LIN {X 0.214,Y -702.984,Z 640.438,A 0.000,B 0.000,C 90.000,E1 294.847} C_DIS
LIN {X -0.283,Y -702.330,Z 640.438,A 0.000,B 0.000,C 90.000,E1 294.771} C_DIS
LIN {X 0.270,Y -699.025,Z 640.435,A 0.000,B 0.000,C 90.000,E1 294.259} C_DIS
LIN {X 0.118,Y -697.927,Z 640.434,A 0.000,B 0.000,C 90.000,E1 294.155} C_DIS
LIN {X 0.250,Y -696.247,Z 640.434,A 0.000,B 0.000,C 90.000,E1 294.027} C_DIS
LIN {X 0.435,Y -691.769,Z 640.433,A 0.000,B 0.000,C 90.000,E1 293.823} C_DIS
LIN {X 0.326,Y -685.920,Z 640.432,A 0.000,B 0.000,C 90.000,E1 293.643} C_DIS
LIN {X -0.028,Y -681.507,Z 640.431,A 0.000,B 0.000,C 90.000,E1 293.567} C_DIS
LIN {X -0.084,Y -673.236,Z 640.430,A 0.000,B 0.000,C 90.000,E1 293.462} C_DIS
LIN {X 0.101,Y -666.043,Z 640.430,A 0.000,B 0.000,C 90.000,E1 293.387} C_DIS
LIN {X 0.093,Y -649.725,Z 640.429,A 0.000,B 0.000,C 90.000,E1 293.153} C_DIS
LIN {X -0.148,Y -639.864,Z 640.428,A 0.000,B 0.000,C 90.000,E1 293.003} C_DIS
LIN {X 0.048,Y -630.020,Z 640.427,A 0.000,B 0.000,C 90.000,E1 292.770} C_DIS
LIN {X -0.345,Y -616.725,Z 640.425,A 0.000,B 0.000,C 90.000,E1 292.461} C_DIS
LIN {X 0.086,Y -589.337,Z 640.420,A 0.000,B 0.000,C 90.000,E1 291.589} C_DIS
LIN {X -0.163,Y -576.913,Z 640.418,A 0.000,B 0.000,C 90.000,E1 291.227} C_DIS
LIN {X -0.001,Y -564.499,Z 640.416,A 0.000,B 0.000,C 90.000,E1 290.844} C_DIS
LIN {X 0.289,Y -559.704,Z 640.415,A 0.000,B 0.000,C 90.000,E1 290.610} C_DIS
LIN {X 0.143,Y -556.813,Z 640.414,A 0.000,B 0.000,C 90.000,E1 290.429} C_DIS
LIN {X 0.112,Y -556.775,Z 640.414,A 0.000,B 0.000,C 90.000,E1 290.429} C_DIS
LIN {X -0.163,Y -556.015,Z 640.412,A 0.000,B 0.000,C 90.000,E1 290.248} C_DIS
LIN {X 0.014,Y -555.587,Z 640.410,A 0.000,B 0.000,C 90.000,E1 289.812} C_DIS
LIN {X -0.233,Y -555.561,Z 640.404,A 0.000,B 0.000,C 90.000,E1 288.725} C_DIS
LIN {X -0.215,Y -555.366,Z 640.396,A 0.000,B 0.000,C 90.000,E1 287.330} C_DIS
LIN {X -0.115,Y -555.080,Z 640.390,A 0.000,B 0.000,C 90.000,E1 286.205} C_DIS
LIN {X 0.258,Y -554.527,Z 640.382,A 0.000,B 0.000,C 90.000,E1 284.773} C_DIS
LIN {X -0.065,Y -553.860,Z 640.375,A 0.000,B 0.000,C 90.000,E1 283.411} C_DIS
LIN {X 0.136,Y -552.938,Z 640.365,A 0.000,B 0.000,C 90.000,E1 281.715} C_DIS
LIN {X 0.079,Y -552.458,Z 640.359,A 0.000,B 0.000,C 90.000,E1 280.602} C_DIS
LIN {X 0.264,Y -551.690,Z 640.348,A 0.000,B 0.000,C 90.000,E1 278.624} C_DIS
LIN {X -0.277,Y -550.949,Z 640.337,A 0.000,B 0.000,C 90.000,E1 276.720} C_DIS
LIN {X 0.258,Y -550.396,Z 640.326,A 0.000,B 0.000,C 90.000,E1 274.702} C_DIS
LIN {X 0.000,Y -550.065,Z 640.319,A 0.000,B 0.000,C 90.000,E1 273.326} C_DIS
LIN {X -0.182,Y -549.599,Z 640.309,A 0.000,B 0.000,C 90.000,E1 271.661} C_DIS
LIN {X 0.139,Y -549.034,Z 640.300,A 0.000,B 0.000,C 90.000,E1 269.943} C_DIS
LIN {X -0.153,Y -548.291,Z 640.292,A 0.000,B 0.000,C 90.000,E1 268.568} C_DIS
LIN {X 0.101,Y -547.676,Z 640.284,A 0.000,B 0.000,C 90.000,E1 267.135} C_DIS
LIN {X -0.168,Y -546.950,Z 640.276,A 0.000,B 0.000,C 90.000,E1 265.755} C_DIS
LIN {X 0.100,Y -545.943,Z 640.269,A 0.000,B 0.000,C 90.000,E1 264.318} C_DIS
LIN {X -0.140,Y -544.897,Z 640.261,A 0.000,B 0.000,C 90.000,E1 262.932} C_DIS
LIN {X 0.057,Y -543.716,Z 640.254,A 0.000,B 0.000,C 90.000,E1 261.781} C_DIS
LIN {X 0.013,Y -541.556,Z 640.243,A 0.000,B 0.000,C 90.000,E1 259.803} C_DIS
LIN {X -0.159,Y -540.004,Z 640.234,A 0.000,B 0.000,C 90.000,E1 258.117} C_DIS
LIN {X -0.015,Y -538.115,Z 640.221,A 0.000,B 0.000,C 90.000,E1 255.825} C_DIS
LIN {X -0.019,Y -537.132,Z 640.215,A 0.000,B 0.000,C 90.000,E1 254.685} C_DIS
LIN {X -0.173,Y -535.984,Z 640.209,A 0.000,B 0.000,C 90.000,E1 253.559} C_DIS
LIN {X -0.230,Y -533.804,Z 640.196,A 0.000,B 0.000,C 90.000,E1 251.275} C_DIS
LIN {X 0.193,Y -532.904,Z 640.191,A 0.000,B 0.000,C 90.000,E1 250.369} C_DIS
LIN {X -0.201,Y -531.346,Z 640.185,A 0.000,B 0.000,C 90.000,E1 249.263} C_DIS
LIN {X 0.066,Y -529.285,Z 640.177,A 0.000,B 0.000,C 90.000,E1 247.794} C_DIS
LIN {X -0.176,Y -527.436,Z 640.170,A 0.000,B 0.000,C 90.000,E1 246.666} C_DIS
LIN {X -0.130,Y -525.978,Z 640.165,A 0.000,B 0.000,C 90.000,E1 245.793} C_DIS
LIN {X 0.280,Y -523.709,Z 640.159,A 0.000,B 0.000,C 90.000,E1 244.588} C_DIS
LIN {X -0.047,Y -521.275,Z 640.153,A 0.000,B 0.000,C 90.000,E1 243.461} C_DIS
LIN {X 0.187,Y -518.199,Z 640.144,A 0.000,B 0.000,C 90.000,E1 241.975} C_DIS
LIN {X -0.092,Y -515.078,Z 640.136,A 0.000,B 0.000,C 90.000,E1 240.539} C_DIS
LIN {X 0.182,Y -512.332,Z 640.130,A 0.000,B 0.000,C 90.000,E1 239.331} C_DIS
LIN {X -0.046,Y -508.136,Z 640.120,A 0.000,B 0.000,C 90.000,E1 237.582} C_DIS
LIN {X 0.015,Y -504.589,Z 640.112,A 0.000,B 0.000,C 90.000,E1 236.087} C_DIS
LIN {X -0.013,Y -501.554,Z 640.105,A 0.000,B 0.000,C 90.000,E1 234.895} C_DIS
LIN {X -0.083,Y -498.368,Z 640.098,A 0.000,B 0.000,C 90.000,E1 233.703} C_DIS
LIN {X 0.072,Y -491.532,Z 640.083,A 0.000,B 0.000,C 90.000,E1 230.964} C_DIS
LIN {X 0.058,Y -487.091,Z 640.073,A 0.000,B 0.000,C 90.000,E1 229.138} C_DIS
LIN {X -0.113,Y -481.191,Z 640.059,A 0.000,B 0.000,C 90.000,E1 226.701} C_DIS
LIN {X 0.054,Y -478.156,Z 640.053,A 0.000,B 0.000,C 90.000,E1 225.445} C_DIS
LIN {X 0.278,Y -474.467,Z 640.044,A 0.000,B 0.000,C 90.000,E1 223.866} C_DIS
LIN {X -0.233,Y -470.885,Z 640.035,A 0.000,B 0.000,C 90.000,E1 222.366} C_DIS
LIN {X 0.140,Y -465.420,Z 640.021,A 0.000,B 0.000,C 90.000,E1 219.806} C_DIS
LIN {X -0.098,Y -461.340,Z 640.011,A 0.000,B 0.000,C 90.000,E1 217.935} C_DIS
LIN {X -0.151,Y -456.212,Z 639.997,A 0.000,B 0.000,C 90.000,E1 215.391} C_DIS
LIN {X -0.138,Y -453.326,Z 639.988,A 0.000,B 0.000,C 90.000,E1 213.785} C_DIS
LIN {X -0.101,Y -448.042,Z 639.971,A 0.000,B 0.000,C 90.000,E1 210.875} C_DIS
LIN {X 0.105,Y -444.631,Z 639.961,A 0.000,B 0.000,C 90.000,E1 208.899} C_DIS
LIN {X 0.018,Y -441.087,Z 639.950,A 0.000,B 0.000,C 90.000,E1 206.950} C_DIS
LIN {X -0.030,Y -438.709,Z 639.943,A 0.000,B 0.000,C 90.000,E1 205.643} C_DIS
LIN {X 0.136,Y -435.079,Z 639.932,A 0.000,B 0.000,C 90.000,E1 203.643} C_DIS
LIN {X 0.014,Y -432.764,Z 639.924,A 0.000,B 0.000,C 90.000,E1 202.333} C_DIS
LIN {X 0.086,Y -428.719,Z 639.911,A 0.000,B 0.000,C 90.000,E1 199.993} C_DIS
LIN {X 0.156,Y -424.805,Z 639.898,A 0.000,B 0.000,C 90.000,E1 197.638} C_DIS
LIN {X -0.188,Y -421.615,Z 639.887,A 0.000,B 0.000,C 90.000,E1 195.662} C_DIS
LIN {X 0.035,Y -418.916,Z 639.878,A 0.000,B 0.000,C 90.000,E1 193.939} C_DIS
LIN {X 0.058,Y -415.763,Z 639.866,A 0.000,B 0.000,C 90.000,E1 191.895} C_DIS
LIN {X 0.058,Y -412.228,Z 639.853,A 0.000,B 0.000,C 90.000,E1 189.500} C_DIS
LIN {X 0.200,Y -410.259,Z 639.845,A 0.000,B 0.000,C 90.000,E1 188.106} C_DIS
LIN {X -0.151,Y -406.790,Z 639.832,A 0.000,B 0.000,C 90.000,E1 185.739} C_DIS
LIN {X 0.128,Y -403.391,Z 639.816,A 0.000,B 0.000,C 90.000,E1 182.922} C_DIS
LIN {X -0.036,Y -398.663,Z 639.789,A 0.000,B 0.000,C 90.000,E1 178.051} C_DIS
LIN {X 0.172,Y -396.253,Z 639.766,A 0.000,B 0.000,C 90.000,E1 173.799} C_DIS
LIN {X -0.114,Y -395.651,Z 639.754,A 0.000,B 0.000,C 90.000,E1 171.724} C_DIS
LIN {X 0.123,Y -395.202,Z 639.740,A 0.000,B 0.000,C 90.000,E1 169.218} C_DIS
LIN {X 0.025,Y -395.157,Z 639.721,A 0.000,B 0.000,C 90.000,E1 165.700} C_DIS
LIN {X -0.195,Y -395.441,Z 639.705,A 0.000,B 0.000,C 90.000,E1 162.906} C_DIS
LIN {X 0.192,Y -395.870,Z 639.693,A 0.000,B 0.000,C 90.000,E1 160.732} C_DIS
LIN {X -0.020,Y -396.318,Z 639.681,A 0.000,B 0.000,C 90.000,E1 158.646} C_DIS
LIN {X -0.012,Y -396.971,Z 639.668,A 0.000,B 0.000,C 90.000,E1 156.177} C_DIS
LIN {X -0.041,Y -397.593,Z 639.654,A 0.000,B 0.000,C 90.000,E1 153.717} C_DIS
LIN {X 0.066,Y -398.150,Z 639.642,A 0.000,B 0.000,C 90.000,E1 151.591} C_DIS
LIN {X -0.197,Y -398.673,Z 639.633,A 0.000,B 0.000,C 90.000,E1 149.871} C_DIS
LIN {X -0.023,Y -399.254,Z 639.621,A 0.000,B 0.000,C 90.000,E1 147.740} C_DIS
LIN {X 0.140,Y -400.146,Z 639.607,A 0.000,B 0.000,C 90.000,E1 145.261} C_DIS
LIN {X -0.212,Y -401.026,Z 639.596,A 0.000,B 0.000,C 90.000,E1 143.210} C_DIS
LIN {X -0.176,Y -401.737,Z 639.586,A 0.000,B 0.000,C 90.000,E1 141.457} C_DIS
LIN {X 0.132,Y -402.461,Z 639.576,A 0.000,B 0.000,C 90.000,E1 139.666} C_DIS
LIN {X 0.149,Y -403.113,Z 639.566,A 0.000,B 0.000,C 90.000,E1 137.919} C_DIS
LIN {X -0.008,Y -403.916,Z 639.555,A 0.000,B 0.000,C 90.000,E1 135.850} C_DIS
LIN {X -0.042,Y -404.957,Z 639.541,A 0.000,B 0.000,C 90.000,E1 133.419} C_DIS
LIN {X 0.105,Y -406.638,Z 639.526,A 0.000,B 0.000,C 90.000,E1 130.620} C_DIS
LIN {X 0.078,Y -407.304,Z 639.522,A 0.000,B 0.000,C 90.000,E1 129.930} C_DIS
LIN {X 0.029,Y -408.620,Z 639.517,A 0.000,B 0.000,C 90.000,E1 129.072} C_DIS
LIN {X 0.015,Y -410.546,Z 639.513,A 0.000,B 0.000,C 90.000,E1 128.382} C_DIS
LIN {X -0.069,Y -411.560,Z 639.512,A 0.000,B 0.000,C 90.000,E1 128.222} C_DIS
LIN {X -0.162,Y -413.181,Z 639.510,A 0.000,B 0.000,C 90.000,E1 127.890} C_DIS
LIN {X 0.099,Y -416.926,Z 639.508,A 0.000,B 0.000,C 90.000,E1 127.443} C_DIS
LIN {X -0.118,Y -420.836,Z 639.506,A 0.000,B 0.000,C 90.000,E1 127.156} C_DIS
LIN {X 0.057,Y -442.467,Z 639.499,A 0.000,B 0.000,C 90.000,E1 125.724} C_DIS
LIN {X -0.069,Y -450.784,Z 639.496,A 0.000,B 0.000,C 90.000,E1 125.231} C_DIS
LIN {X -0.113,Y -460.538,Z 639.492,A 0.000,B 0.000,C 90.000,E1 124.612} C_DIS
LIN {X 0.212,Y -473.139,Z 639.487,A 0.000,B 0.000,C 90.000,E1 123.706} C_DIS
LIN {X -0.040,Y -480.978,Z 639.484,A 0.000,B 0.000,C 90.000,E1 123.166} C_DIS
LIN {X -0.212,Y -488.438,Z 639.481,A 0.000,B 0.000,C 90.000,E1 122.625} C_DIS
LIN {X -0.011,Y -496.000,Z 639.478,A 0.000,B 0.000,C 90.000,E1 122.005} C_DIS
LIN {X -0.106,Y -505.725,Z 639.473,A 0.000,B 0.000,C 90.000,E1 121.209} C_DIS
LIN {X -0.173,Y -512.904,Z 639.470,A 0.000,B 0.000,C 90.000,E1 120.590} C_DIS
LIN {X -0.071,Y -518.358,Z 639.467,A 0.000,B 0.000,C 90.000,E1 120.079} C_DIS
LIN {X -0.102,Y -524.925,Z 639.464,A 0.000,B 0.000,C 90.000,E1 119.461} C_DIS
LIN {X 0.099,Y -531.758,Z 639.460,A 0.000,B 0.000,C 90.000,E1 118.771} C_DIS
LIN {X 0.053,Y -536.831,Z 639.457,A 0.000,B 0.000,C 90.000,E1 118.231} C_DIS
LIN {X -0.113,Y -541.360,Z 639.454,A 0.000,B 0.000,C 90.000,E1 117.719} C_DIS
LIN {X -0.071,Y -546.495,Z 639.450,A 0.000,B 0.000,C 90.000,E1 117.052} C_DIS
LIN {X -0.077,Y -550.302,Z 639.447,A 0.000,B 0.000,C 90.000,E1 116.488} C_DIS
LIN {X -0.163,Y -554.583,Z 639.443,A 0.000,B 0.000,C 90.000,E1 115.796} C_DIS
LIN {X -0.078,Y -559.013,Z 639.439,A 0.000,B 0.000,C 90.000,E1 114.951} C_DIS
LIN {X -0.189,Y -562.959,Z 639.434,A 0.000,B 0.000,C 90.000,E1 114.131} C_DIS
LIN {X 0.258,Y -566.594,Z 639.429,A 0.000,B 0.000,C 90.000,E1 113.259} C_DIS
LIN {X -0.001,Y -569.978,Z 639.425,A 0.000,B 0.000,C 90.000,E1 112.461} C_DIS
LIN {X 0.140,Y -573.938,Z 639.419,A 0.000,B 0.000,C 90.000,E1 111.354} C_DIS
LIN {X 0.333,Y -575.783,Z 639.416,A 0.000,B 0.000,C 90.000,E1 110.791} C_DIS
LIN {X 0.172,Y -578.288,Z 639.411,A 0.000,B 0.000,C 90.000,E1 109.993} C_DIS
LIN {X 0.227,Y -581.303,Z 639.405,A 0.000,B 0.000,C 90.000,E1 108.906} C_DIS
LIN {X -0.067,Y -583.345,Z 639.401,A 0.000,B 0.000,C 90.000,E1 108.127} C_DIS
LIN {X -0.266,Y -586.358,Z 639.393,A 0.000,B 0.000,C 90.000,E1 106.804} C_DIS
LIN {X -0.076,Y -591.364,Z 639.381,A 0.000,B 0.000,C 90.000,E1 104.647} C_DIS
LIN {X 0.099,Y -595.831,Z 639.371,A 0.000,B 0.000,C 90.000,E1 102.771} C_DIS
LIN {X -0.203,Y -598.908,Z 639.364,A 0.000,B 0.000,C 90.000,E1 101.478} C_DIS
LIN {X 0.017,Y -602.053,Z 639.356,A 0.000,B 0.000,C 90.000,E1 100.141} C_DIS
LIN {X -0.301,Y -605.007,Z 639.349,A 0.000,B 0.000,C 90.000,E1 98.859} C_DIS
LIN {X 0.295,Y -607.255,Z 639.343,A 0.000,B 0.000,C 90.000,E1 97.757} C_DIS
LIN {X -0.039,Y -609.837,Z 639.336,A 0.000,B 0.000,C 90.000,E1 96.486} C_DIS
LIN {X -0.124,Y -612.554,Z 639.327,A 0.000,B 0.000,C 90.000,E1 94.935} C_DIS
LIN {X 0.176,Y -614.578,Z 639.320,A 0.000,B 0.000,C 90.000,E1 93.612} C_DIS
LIN {X -0.146,Y -616.328,Z 639.313,A 0.000,B 0.000,C 90.000,E1 92.350} C_DIS
LIN {X -0.133,Y -617.527,Z 639.307,A 0.000,B 0.000,C 90.000,E1 91.318} C_DIS
LIN {X -0.112,Y -618.745,Z 639.299,A 0.000,B 0.000,C 90.000,E1 89.771} C_DIS
LIN {X -0.085,Y -619.350,Z 639.293,A 0.000,B 0.000,C 90.000,E1 88.740} C_DIS
LIN {X -0.033,Y -619.644,Z 639.287,A 0.000,B 0.000,C 90.000,E1 87.707} C_DIS
LIN {X -0.321,Y -619.669,Z 639.283,A 0.000,B 0.000,C 90.000,E1 86.963} C_DIS
LIN {X -0.224,Y -619.534,Z 639.277,A 0.000,B 0.000,C 90.000,E1 85.927} C_DIS
LIN {X -0.168,Y -619.186,Z 639.272,A 0.000,B 0.000,C 90.000,E1 84.894} C_DIS
LIN {X 0.233,Y -618.474,Z 639.264,A 0.000,B 0.000,C 90.000,E1 83.571} C_DIS
LIN {X -0.292,Y -617.789,Z 639.259,A 0.000,B 0.000,C 90.000,E1 82.591} C_DIS
LIN {X 0.114,Y -617.072,Z 639.254,A 0.000,B 0.000,C 90.000,E1 81.781} C_DIS
LIN {X 0.268,Y -615.828,Z 639.249,A 0.000,B 0.000,C 90.000,E1 80.735} C_DIS
LIN {X 0.163,Y -614.044,Z 639.242,A 0.000,B 0.000,C 90.000,E1 79.454} C_DIS
LIN {X 0.025,Y -611.983,Z 639.234,A 0.000,B 0.000,C 90.000,E1 78.173} C_DIS
LIN {X -0.025,Y -609.699,Z 639.227,A 0.000,B 0.000,C 90.000,E1 76.881} C_DIS
LIN {X 0.140,Y -607.779,Z 639.221,A 0.000,B 0.000,C 90.000,E1 75.825} C_DIS
LIN {X 0.161,Y -605.161,Z 639.214,A 0.000,B 0.000,C 90.000,E1 74.519} C_DIS
LIN {X -0.169,Y -602.830,Z 639.208,A 0.000,B 0.000,C 90.000,E1 73.504} C_DIS
LIN {X -0.058,Y -599.843,Z 639.201,A 0.000,B 0.000,C 90.000,E1 72.181} C_DIS
LIN {X 0.295,Y -597.192,Z 639.195,A 0.000,B 0.000,C 90.000,E1 71.094} C_DIS
LIN {X 0.046,Y -594.117,Z 639.189,A 0.000,B 0.000,C 90.000,E1 70.061} C_DIS
LIN {X 0.074,Y -591.600,Z 639.185,A 0.000,B 0.000,C 90.000,E1 69.263} C_DIS
LIN {X 0.078,Y -588.849,Z 639.180,A 0.000,B 0.000,C 90.000,E1 68.465} C_DIS
LIN {X -0.072,Y -584.716,Z 639.174,A 0.000,B 0.000,C 90.000,E1 67.411} C_DIS
LIN {X -0.277,Y -580.359,Z 639.169,A 0.000,B 0.000,C 90.000,E1 66.357} C_DIS
LIN {X 0.063,Y -574.233,Z 639.161,A 0.000,B 0.000,C 90.000,E1 64.973} C_DIS
LIN {X 0.268,Y -571.589,Z 639.158,A 0.000,B 0.000,C 90.000,E1 64.409} C_DIS
LIN {X -0.063,Y -568.759,Z 639.155,A 0.000,B 0.000,C 90.000,E1 63.896} C_DIS
LIN {X 0.005,Y -564.884,Z 639.151,A 0.000,B 0.000,C 90.000,E1 63.204} C_DIS
LIN {X -0.112,Y -561.591,Z 639.148,A 0.000,B 0.000,C 90.000,E1 62.666} C_DIS
LIN {X 0.097,Y -557.022,Z 639.144,A 0.000,B 0.000,C 90.000,E1 61.975} C_DIS
LIN {X -0.062,Y -553.002,Z 639.141,A 0.000,B 0.000,C 90.000,E1 61.435} C_DIS
LIN {X 0.088,Y -549.418,Z 639.139,A 0.000,B 0.000,C 90.000,E1 61.001} C_DIS
LIN {X 0.124,Y -547.052,Z 639.137,A 0.000,B 0.000,C 90.000,E1 60.717} C_DIS
LIN {X -0.069,Y -543.497,Z 639.135,A 0.000,B 0.000,C 90.000,E1 60.333} C_DIS
LIN {X 0.302,Y -538.237,Z 639.132,A 0.000,B 0.000,C 90.000,E1 59.793} C_DIS
LIN {X -0.209,Y -533.738,Z 639.130,A 0.000,B 0.000,C 90.000,E1 59.459} C_DIS
LIN {X -0.199,Y -527.676,Z 639.128,A 0.000,B 0.000,C 90.000,E1 58.997} C_DIS
LIN {X 0.158,Y -521.319,Z 639.125,A 0.000,B 0.000,C 90.000,E1 58.535} C_DIS
LIN {X 0.023,Y -516.351,Z 639.124,A 0.000,B 0.000,C 90.000,E1 58.250} C_DIS
LIN {X 0.258,Y -506.211,Z 639.121,A 0.000,B 0.000,C 90.000,E1 57.661} C_DIS
LIN {X -0.156,Y -482.576,Z 639.114,A 0.000,B 0.000,C 90.000,E1 56.501} C_DIS
LIN {X 0.027,Y -460.468,Z 639.108,A 0.000,B 0.000,C 90.000,E1 55.341} C_DIS
LIN {X 0.094,Y -438.216,Z 639.101,A 0.000,B 0.000,C 90.000,E1 54.116} C_DIS
LIN {X 0.050,Y -438.150,Z 639.101,A 0.000,B 0.000,C 90.000,E1 54.116} C_DIS
LIN {X -0.079,Y -431.839,Z 639.083,A 0.000,B 0.000,C 90.000,E1 51.009} C_DIS
LIN {X 0.180,Y -431.143,Z 639.082,A 0.000,B 0.000,C 90.000,E1 50.642} C_DIS
LIN {X 0.111,Y -423.698,Z 639.064,A 0.000,B 0.000,C 90.000,E1 47.472} C_DIS
LIN {X 0.080,Y -424.089,Z 639.057,A 0.000,B 0.000,C 90.000,E1 46.296} C_DIS
LIN {X -0.206,Y -424.329,Z 639.052,A 0.000,B 0.000,C 90.000,E1 45.324} C_DIS
LIN {X -0.052,Y -424.762,Z 639.037,A 0.000,B 0.000,C 90.000,E1 42.609} C_DIS
LIN {X -0.275,Y -425.406,Z 639.026,A 0.000,B 0.000,C 90.000,E1 40.620} C_DIS
LIN {X 0.064,Y -426.388,Z 639.012,A 0.000,B 0.000,C 90.000,E1 38.222} C_DIS
LIN {X -0.003,Y -427.318,Z 639.001,A 0.000,B 0.000,C 90.000,E1 36.217} C_DIS
LIN {X -0.167,Y -428.037,Z 638.994,A 0.000,B 0.000,C 90.000,E1 34.898} C_DIS
LIN {X -0.094,Y -428.902,Z 638.983,A 0.000,B 0.000,C 90.000,E1 32.880} C_DIS
LIN {X -0.104,Y -429.733,Z 638.971,A 0.000,B 0.000,C 90.000,E1 30.875} C_DIS
LIN {X -0.096,Y -430.417,Z 638.962,A 0.000,B 0.000,C 90.000,E1 29.205} C_DIS
LIN {X 0.085,Y -431.164,Z 638.953,A 0.000,B 0.000,C 90.000,E1 27.513} C_DIS
LIN {X -0.104,Y -432.164,Z 638.942,A 0.000,B 0.000,C 90.000,E1 25.540} C_DIS
LIN {X 0.122,Y -433.288,Z 638.931,A 0.000,B 0.000,C 90.000,E1 23.515} C_DIS
LIN {X 0.029,Y -434.557,Z 638.920,A 0.000,B 0.000,C 90.000,E1 21.535} C_DIS
LIN {X -0.020,Y -435.592,Z 638.911,A 0.000,B 0.000,C 90.000,E1 19.885} C_DIS
LIN {X 0.188,Y -436.754,Z 638.899,A 0.000,B 0.000,C 90.000,E1 17.873} C_DIS
LIN {X -0.149,Y -438.145,Z 638.887,A 0.000,B 0.000,C 90.000,E1 15.607} C_DIS
LIN {X 0.109,Y -440.016,Z 638.872,A 0.000,B 0.000,C 90.000,E1 12.939} C_DIS
LIN {X -0.030,Y -441.896,Z 638.859,A 0.000,B 0.000,C 90.000,E1 10.658} C_DIS
LIN {X 0.067,Y -444.666,Z 638.843,A 0.000,B 0.000,C 90.000,E1 7.701} C_DIS
LIN {X 0.111,Y -446.688,Z 638.832,A 0.000,B 0.000,C 90.000,E1 5.739} C_DIS
LIN {X 0.180,Y -450.113,Z 638.816,A 0.000,B 0.000,C 90.000,E1 2.808} C_DIS
LIN {X -0.199,Y -452.588,Z 638.805,A 0.000,B 0.000,C 90.000,E1 0.917} C_DIS
LIN {X 0.163,Y -456.504,Z 638.790,A 0.000,B 0.000,C 90.000,E1 358.165} C_DIS
LIN {X 0.204,Y -459.105,Z 638.781,A 0.000,B 0.000,C 90.000,E1 356.560} C_DIS
LIN {X 0.055,Y -462.306,Z 638.770,A 0.000,B 0.000,C 90.000,E1 354.666} C_DIS
LIN {X 0.063,Y -465.626,Z 638.760,A 0.000,B 0.000,C 90.000,E1 352.761} C_DIS
LIN {X 0.217,Y -468.922,Z 638.749,A 0.000,B 0.000,C 90.000,E1 350.849} C_DIS
LIN {X -0.132,Y -471.112,Z 638.742,A 0.000,B 0.000,C 90.000,E1 349.634} C_DIS
LIN {X 0.148,Y -474.860,Z 638.730,A 0.000,B 0.000,C 90.000,E1 347.409} C_DIS
LIN {X 0.020,Y -479.405,Z 638.716,A 0.000,B 0.000,C 90.000,E1 344.936} C_DIS
LIN {X -0.192,Y -484.083,Z 638.703,A 0.000,B 0.000,C 90.000,E1 342.489} C_DIS
LIN {X 0.159,Y -487.675,Z 638.692,A 0.000,B 0.000,C 90.000,E1 340.604} C_DIS
LIN {X 0.111,Y -490.671,Z 638.684,A 0.000,B 0.000,C 90.000,E1 339.082} C_DIS
LIN {X 0.252,Y -493.055,Z 638.677,A 0.000,B 0.000,C 90.000,E1 337.847} C_DIS
LIN {X -0.074,Y -494.653,Z 638.672,A 0.000,B 0.000,C 90.000,E1 336.975} C_DIS
LIN {X -0.281,Y -497.144,Z 638.664,A 0.000,B 0.000,C 90.000,E1 335.485} C_DIS
LIN {X 0.031,Y -499.972,Z 638.654,A 0.000,B 0.000,C 90.000,E1 333.640} C_DIS
LIN {X -0.044,Y -502.754,Z 638.644,A 0.000,B 0.000,C 90.000,E1 331.847} C_DIS
LIN {X 0.198,Y -508.652,Z 638.625,A 0.000,B 0.000,C 90.000,E1 328.535} C_DIS
LIN {X 0.054,Y -510.798,Z 638.620,A 0.000,B 0.000,C 90.000,E1 327.661} C_DIS
LIN {X 0.298,Y -512.682,Z 638.617,A 0.000,B 0.000,C 90.000,E1 327.041} C_DIS
LIN {X -0.155,Y -515.106,Z 638.614,A 0.000,B 0.000,C 90.000,E1 326.501} C_DIS
LIN {X 0.306,Y -517.597,Z 638.611,A 0.000,B 0.000,C 90.000,E1 326.008} C_DIS
LIN {X 0.062,Y -520.974,Z 638.609,A 0.000,B 0.000,C 90.000,E1 325.595} C_DIS
LIN {X 0.192,Y -523.917,Z 638.607,A 0.000,B 0.000,C 90.000,E1 325.261} C_DIS
LIN {X 0.257,Y -530.298,Z 638.604,A 0.000,B 0.000,C 90.000,E1 324.689} C_DIS
LIN {X -0.225,Y -547.687,Z 638.596,A 0.000,B 0.000,C 90.000,E1 323.336} C_DIS
LIN {X -0.048,Y -556.154,Z 638.592,A 0.000,B 0.000,C 90.000,E1 322.603} C_DIS
LIN {X 0.167,Y -567.400,Z 638.587,A 0.000,B 0.000,C 90.000,E1 321.618} C_DIS
LIN {X 0.174,Y -579.786,Z 638.581,A 0.000,B 0.000,C 90.000,E1 320.517} C_DIS
LIN {X 0.169,Y -590.603,Z 638.575,A 0.000,B 0.000,C 90.000,E1 319.542} C_DIS
LIN {X 0.208,Y -599.582,Z 638.571,A 0.000,B 0.000,C 90.000,E1 318.690} C_DIS
LIN {X 0.147,Y -603.451,Z 638.569,A 0.000,B 0.000,C 90.000,E1 318.324} C_DIS
LIN {X -0.384,Y -611.958,Z 638.564,A 0.000,B 0.000,C 90.000,E1 317.472} C_DIS
LIN {X 0.089,Y -617.498,Z 638.560,A 0.000,B 0.000,C 90.000,E1 316.782} C_DIS
LIN {X 0.044,Y -620.550,Z 638.558,A 0.000,B 0.000,C 90.000,E1 316.419} C_DIS
LIN {X 0.378,Y -626.351,Z 638.554,A 0.000,B 0.000,C 90.000,E1 315.648} C_DIS
LIN {X 0.004,Y -632.030,Z 638.550,A 0.000,B 0.000,C 90.000,E1 314.919} C_DIS
LIN {X -0.319,Y -637.451,Z 638.545,A 0.000,B 0.000,C 90.000,E1 314.190} C_DIS
LIN {X -0.209,Y -644.470,Z 638.540,A 0.000,B 0.000,C 90.000,E1 313.176} C_DIS
LIN {X 0.071,Y -648.686,Z 638.536,A 0.000,B 0.000,C 90.000,E1 312.528} C_DIS
LIN {X -0.016,Y -651.957,Z 638.534,A 0.000,B 0.000,C 90.000,E1 312.043} C_DIS
LIN {X -0.098,Y -656.684,Z 638.529,A 0.000,B 0.000,C 90.000,E1 311.310} C_DIS
LIN {X -0.158,Y -660.324,Z 638.526,A 0.000,B 0.000,C 90.000,E1 310.701} C_DIS
LIN {X 0.267,Y -664.285,Z 638.522,A 0.000,B 0.000,C 90.000,E1 309.930} C_DIS
LIN {X -0.197,Y -666.771,Z 638.519,A 0.000,B 0.000,C 90.000,E1 309.483} C_DIS
LIN {X -0.142,Y -670.151,Z 638.515,A 0.000,B 0.000,C 90.000,E1 308.749} C_DIS
LIN {X 0.062,Y -674.214,Z 638.510,A 0.000,B 0.000,C 90.000,E1 307.764} C_DIS
LIN {X 0.195,Y -676.940,Z 638.506,A 0.000,B 0.000,C 90.000,E1 307.030} C_DIS
LIN {X -0.046,Y -680.209,Z 638.501,A 0.000,B 0.000,C 90.000,E1 306.091} C_DIS
LIN {X 0.303,Y -683.353,Z 638.495,A 0.000,B 0.000,C 90.000,E1 305.105} C_DIS
LIN {X -0.056,Y -687.653,Z 638.487,A 0.000,B 0.000,C 90.000,E1 303.706} C_DIS
LIN {X 0.001,Y -690.328,Z 638.482,A 0.000,B 0.000,C 90.000,E1 302.752} C_DIS
LIN {X -0.265,Y -693.426,Z 638.475,A 0.000,B 0.000,C 90.000,E1 301.592} C_DIS
LIN {X 0.100,Y -695.821,Z 638.470,A 0.000,B 0.000,C 90.000,E1 300.620} C_DIS
LIN {X -0.094,Y -698.544,Z 638.464,A 0.000,B 0.000,C 90.000,E1 299.461} C_DIS
LIN {X 0.351,Y -700.491,Z 638.458,A 0.000,B 0.000,C 90.000,E1 298.487} C_DIS
LIN {X -0.123,Y -702.298,Z 638.453,A 0.000,B 0.000,C 90.000,E1 297.590} C_DIS
LIN {X 0.092,Y -703.480,Z 638.449,A 0.000,B 0.000,C 90.000,E1 296.873} C_DIS
LIN {X 0.001,Y -704.295,Z 638.445,A 0.000,B 0.000,C 90.000,E1 296.181} C_DIS
LIN {X -0.059,Y -704.501,Z 638.443,A 0.000,B 0.000,C 90.000,E1 295.720} C_DIS
LIN {X 0.228,Y -704.340,Z 638.442,A 0.000,B 0.000,C 90.000,E1 295.463} C_DIS
LIN {X -0.138,Y -703.279,Z 638.439,A 0.000,B 0.000,C 90.000,E1 295.027} C_DIS
LIN {X 0.146,Y -702.359,Z 638.438,A 0.000,B 0.000,C 90.000,E1 294.771} C_DIS
LIN {X -0.227,Y -699.016,Z 638.435,A 0.000,B 0.000,C 90.000,E1 294.335} C_DIS
LIN {X -0.093,Y -698.007,Z 638.435,A 0.000,B 0.000,C 90.000,E1 294.207} C_DIS
LIN {X 0.040,Y -696.495,Z 638.434,A 0.000,B 0.000,C 90.000,E1 294.079} C_DIS
LIN {X 0.332,Y -694.302,Z 638.433,A 0.000,B 0.000,C 90.000,E1 293.951} C_DIS
LIN {X -0.173,Y -689.748,Z 638.432,A 0.000,B 0.000,C 90.000,E1 293.823} C_DIS
LIN {X -0.084,Y -685.927,Z 638.432,A 0.000,B 0.000,C 90.000,E1 293.695} C_DIS
LIN {X -0.003,Y -681.958,Z 638.431,A 0.000,B 0.000,C 90.000,E1 293.590} C_DIS
LIN {X 0.058,Y -672.967,Z 638.430,A 0.000,B 0.000,C 90.000,E1 293.462} C_DIS
LIN {X 0.228,Y -665.855,Z 638.430,A 0.000,B 0.000,C 90.000,E1 293.387} C_DIS
LIN {X -0.375,Y -649.556,Z 638.429,A 0.000,B 0.000,C 90.000,E1 293.206} C_DIS
LIN {X -0.269,Y -639.725,Z 638.428,A 0.000,B 0.000,C 90.000,E1 293.025} C_DIS
LIN {X 0.175,Y -629.930,Z 638.427,A 0.000,B 0.000,C 90.000,E1 292.770} C_DIS
LIN {X -0.233,Y -616.602,Z 638.425,A 0.000,B 0.000,C 90.000,E1 292.461} C_DIS
LIN {X -0.195,Y -596.132,Z 638.421,A 0.000,B 0.000,C 90.000,E1 291.844} C_DIS
LIN {X -0.051,Y -578.637,Z 638.418,A 0.000,B 0.000,C 90.000,E1 291.280} C_DIS
LIN {X -0.103,Y -564.298,Z 638.416,A 0.000,B 0.000,C 90.000,E1 290.865} C_DIS
LIN {X -0.169,Y -559.577,Z 638.415,A 0.000,B 0.000,C 90.000,E1 290.663} C_DIS
LIN {X 0.132,Y -556.796,Z 638.414,A 0.000,B 0.000,C 90.000,E1 290.429} C_DIS
LIN {X 0.097,Y -556.769,Z 638.414,A 0.000,B 0.000,C 90.000,E1 290.429} C_DIS
LIN {X -0.262,Y -555.974,Z 638.412,A 0.000,B 0.000,C 90.000,E1 290.248} C_DIS
LIN {X 0.212,Y -555.621,Z 638.410,A 0.000,B 0.000,C 90.000,E1 289.812} C_DIS
LIN {X -0.052,Y -555.663,Z 638.404,A 0.000,B 0.000,C 90.000,E1 288.725} C_DIS
LIN {X -0.032,Y -555.489,Z 638.396,A 0.000,B 0.000,C 90.000,E1 287.330} C_DIS
LIN {X 0.070,Y -555.179,Z 638.390,A 0.000,B 0.000,C 90.000,E1 286.205} C_DIS
LIN {X 0.178,Y -554.783,Z 638.384,A 0.000,B 0.000,C 90.000,E1 285.079} C_DIS
LIN {X 0.000,Y -554.133,Z 638.376,A 0.000,B 0.000,C 90.000,E1 283.703} C_DIS
LIN {X 0.079,Y -553.373,Z 638.368,A 0.000,B 0.000,C 90.000,E1 282.299} C_DIS
LIN {X 0.272,Y -552.563,Z 638.359,A 0.000,B 0.000,C 90.000,E1 280.602} C_DIS
LIN {X -0.086,Y -551.792,Z 638.348,A 0.000,B 0.000,C 90.000,E1 278.681} C_DIS
LIN {X -0.120,Y -551.132,Z 638.339,A 0.000,B 0.000,C 90.000,E1 277.004} C_DIS
LIN {X -0.186,Y -550.526,Z 638.328,A 0.000,B 0.000,C 90.000,E1 275.049} C_DIS
LIN {X 0.200,Y -550.101,Z 638.319,A 0.000,B 0.000,C 90.000,E1 273.326} C_DIS
LIN {X -0.052,Y -549.745,Z 638.311,A 0.000,B 0.000,C 90.000,E1 271.949} C_DIS
LIN {X -0.262,Y -549.195,Z 638.302,A 0.000,B 0.000,C 90.000,E1 270.286} C_DIS
LIN {X -0.051,Y -548.685,Z 638.295,A 0.000,B 0.000,C 90.000,E1 269.141} C_DIS
LIN {X -0.241,Y -547.751,Z 638.284,A 0.000,B 0.000,C 90.000,E1 267.192} C_DIS
LIN {X -0.040,Y -547.209,Z 638.278,A 0.000,B 0.000,C 90.000,E1 266.045} C_DIS
LIN {X 0.192,Y -546.471,Z 638.272,A 0.000,B 0.000,C 90.000,E1 264.894} C_DIS
LIN {X -0.016,Y -545.254,Z 638.262,A 0.000,B 0.000,C 90.000,E1 263.223} C_DIS
LIN {X 0.172,Y -544.484,Z 638.258,A 0.000,B 0.000,C 90.000,E1 262.356} C_DIS
LIN {X -0.019,Y -542.628,Z 638.248,A 0.000,B 0.000,C 90.000,E1 260.679} C_DIS
LIN {X 0.057,Y -540.175,Z 638.234,A 0.000,B 0.000,C 90.000,E1 258.117} C_DIS
LIN {X 0.205,Y -538.283,Z 638.221,A 0.000,B 0.000,C 90.000,E1 255.825} C_DIS
LIN {X 0.260,Y -537.008,Z 638.214,A 0.000,B 0.000,C 90.000,E1 254.393} C_DIS
LIN {X -0.169,Y -535.266,Z 638.204,A 0.000,B 0.000,C 90.000,E1 252.725} C_DIS
LIN {X 0.197,Y -533.637,Z 638.194,A 0.000,B 0.000,C 90.000,E1 250.967} C_DIS
LIN {X 0.117,Y -532.640,Z 638.190,A 0.000,B 0.000,C 90.000,E1 250.115} C_DIS
LIN {X 0.222,Y -531.059,Z 638.183,A 0.000,B 0.000,C 90.000,E1 248.954} C_DIS
LIN {X -0.194,Y -529.404,Z 638.177,A 0.000,B 0.000,C 90.000,E1 247.847} C_DIS
LIN {X 0.233,Y -527.074,Z 638.169,A 0.000,B 0.000,C 90.000,E1 246.357} C_DIS
LIN {X -0.207,Y -525.526,Z 638.164,A 0.000,B 0.000,C 90.000,E1 245.537} C_DIS
LIN {X 0.198,Y -523.203,Z 638.158,A 0.000,B 0.000,C 90.000,E1 244.332} C_DIS
LIN {X 0.240,Y -520.131,Z 638.149,A 0.000,B 0.000,C 90.000,E1 242.871} C_DIS
LIN {X 0.000,Y -517.027,Z 638.141,A 0.000,B 0.000,C 90.000,E1 241.435} C_DIS
LIN {X 0.051,Y -514.456,Z 638.135,A 0.000,B 0.000,C 90.000,E1 240.255} C_DIS
LIN {X -0.289,Y -512.397,Z 638.130,A 0.000,B 0.000,C 90.000,E1 239.410} C_DIS
LIN {X 0.185,Y -508.199,Z 638.120,A 0.000,B 0.000,C 90.000,E1 237.582} C_DIS
LIN {X 0.245,Y -504.596,Z 638.112,A 0.000,B 0.000,C 90.000,E1 236.087} C_DIS
LIN {X 0.217,Y -501.543,Z 638.105,A 0.000,B 0.000,C 90.000,E1 234.895} C_DIS
LIN {X 0.020,Y -497.617,Z 638.097,A 0.000,B 0.000,C 90.000,E1 233.417} C_DIS
LIN {X -0.235,Y -490.764,Z 638.082,A 0.000,B 0.000,C 90.000,E1 230.723} C_DIS
LIN {X 0.110,Y -486.303,Z 638.072,A 0.000,B 0.000,C 90.000,E1 228.852} C_DIS
LIN {X 0.107,Y -481.145,Z 638.060,A 0.000,B 0.000,C 90.000,E1 226.701} C_DIS
LIN {X -0.069,Y -478.105,Z 638.053,A 0.000,B 0.000,C 90.000,E1 225.486} C_DIS
LIN {X -0.075,Y -473.665,Z 638.042,A 0.000,B 0.000,C 90.000,E1 223.623} C_DIS
LIN {X -0.021,Y -470.824,Z 638.035,A 0.000,B 0.000,C 90.000,E1 222.366} C_DIS
LIN {X -0.069,Y -466.020,Z 638.023,A 0.000,B 0.000,C 90.000,E1 220.172} C_DIS
LIN {X -0.085,Y -463.308,Z 638.016,A 0.000,B 0.000,C 90.000,E1 218.910} C_DIS
LIN {X -0.165,Y -458.031,Z 638.002,A 0.000,B 0.000,C 90.000,E1 216.377} C_DIS
LIN {X 0.061,Y -453.259,Z 637.988,A 0.000,B 0.000,C 90.000,E1 213.785} C_DIS
LIN {X 0.093,Y -447.985,Z 637.972,A 0.000,B 0.000,C 90.000,E1 210.875} C_DIS
LIN {X -0.092,Y -444.575,Z 637.961,A 0.000,B 0.000,C 90.000,E1 208.949} C_DIS
LIN {X -0.186,Y -441.034,Z 637.950,A 0.000,B 0.000,C 90.000,E1 207.001} C_DIS
LIN {X -0.034,Y -438.667,Z 637.943,A 0.000,B 0.000,C 90.000,E1 205.668} C_DIS
LIN {X -0.085,Y -435.648,Z 637.933,A 0.000,B 0.000,C 90.000,E1 204.027} C_DIS
LIN {X 0.198,Y -432.731,Z 637.924,A 0.000,B 0.000,C 90.000,E1 202.333} C_DIS
LIN {X 0.267,Y -428.685,Z 637.911,A 0.000,B 0.000,C 90.000,E1 199.993} C_DIS
LIN {X -0.070,Y -424.793,Z 637.898,A 0.000,B 0.000,C 90.000,E1 197.692} C_DIS
LIN {X -0.010,Y -421.611,Z 637.887,A 0.000,B 0.000,C 90.000,E1 195.662} C_DIS
LIN {X -0.138,Y -418.429,Z 637.876,A 0.000,B 0.000,C 90.000,E1 193.647} C_DIS
LIN {X 0.010,Y -414.763,Z 637.862,A 0.000,B 0.000,C 90.000,E1 191.243} C_DIS
LIN {X -0.098,Y -411.330,Z 637.849,A 0.000,B 0.000,C 90.000,E1 188.859} C_DIS
LIN {X 0.037,Y -407.826,Z 637.836,A 0.000,B 0.000,C 90.000,E1 186.429} C_DIS
LIN {X -0.089,Y -403.840,Z 637.818,A 0.000,B 0.000,C 90.000,E1 183.326} C_DIS
LIN {X 0.135,Y -401.485,Z 637.807,A 0.000,B 0.000,C 90.000,E1 181.203} C_DIS
LIN {X 0.090,Y -398.442,Z 637.787,A 0.000,B 0.000,C 90.000,E1 177.707} C_DIS
LIN {X -0.118,Y -396.234,Z 637.764,A 0.000,B 0.000,C 90.000,E1 173.514} C_DIS
LIN {X 0.036,Y -395.656,Z 637.752,A 0.000,B 0.000,C 90.000,E1 171.376} C_DIS
LIN {X -0.113,Y -395.286,Z 637.738,A 0.000,B 0.000,C 90.000,E1 168.926} C_DIS
LIN {X -0.168,Y -395.283,Z 637.721,A 0.000,B 0.000,C 90.000,E1 165.755} C_DIS
LIN {X 0.000,Y -395.614,Z 637.705,A 0.000,B 0.000,C 90.000,E1 162.906} C_DIS
LIN {X 0.016,Y -396.015,Z 637.693,A 0.000,B 0.000,C 90.000,E1 160.786} C_DIS
LIN {X -0.026,Y -396.399,Z 637.684,A 0.000,B 0.000,C 90.000,E1 159.028} C_DIS
LIN {X 0.221,Y -396.837,Z 637.674,A 0.000,B 0.000,C 90.000,E1 157.230} C_DIS
LIN {X 0.113,Y -397.298,Z 637.664,A 0.000,B 0.000,C 90.000,E1 155.485} C_DIS
LIN {X 0.042,Y -397.903,Z 637.652,A 0.000,B 0.000,C 90.000,E1 153.384} C_DIS
LIN {X 0.163,Y -398.476,Z 637.641,A 0.000,B 0.000,C 90.000,E1 151.257} C_DIS
LIN {X -0.092,Y -398.987,Z 637.631,A 0.000,B 0.000,C 90.000,E1 149.537} C_DIS
LIN {X -0.247,Y -399.581,Z 637.619,A 0.000,B 0.000,C 90.000,E1 147.454} C_DIS
LIN {X 0.047,Y -400.347,Z 637.607,A 0.000,B 0.000,C 90.000,E1 145.308} C_DIS
LIN {X 0.031,Y -401.222,Z 637.596,A 0.000,B 0.000,C 90.000,E1 143.210} C_DIS
LIN {X 0.070,Y -401.927,Z 637.586,A 0.000,B 0.000,C 90.000,E1 141.457} C_DIS
LIN {X 0.121,Y -402.621,Z 637.576,A 0.000,B 0.000,C 90.000,E1 139.703} C_DIS
LIN {X 0.009,Y -403.118,Z 637.569,A 0.000,B 0.000,C 90.000,E1 138.324} C_DIS
LIN {X 0.131,Y -403.899,Z 637.557,A 0.000,B 0.000,C 90.000,E1 136.215} C_DIS
LIN {X -0.143,Y -404.580,Z 637.547,A 0.000,B 0.000,C 90.000,E1 134.514} C_DIS
LIN {X -0.011,Y -405.882,Z 637.532,A 0.000,B 0.000,C 90.000,E1 131.714} C_DIS
LIN {X 0.080,Y -407.193,Z 637.522,A 0.000,B 0.000,C 90.000,E1 129.967} C_DIS
LIN {X -0.110,Y -408.590,Z 637.516,A 0.000,B 0.000,C 90.000,E1 128.955} C_DIS
LIN {X -0.171,Y -410.677,Z 637.512,A 0.000,B 0.000,C 90.000,E1 128.177} C_DIS
LIN {X -0.012,Y -412.178,Z 637.510,A 0.000,B 0.000,C 90.000,E1 127.810} C_DIS
LIN {X -0.053,Y -412.711,Z 637.510,A 0.000,B 0.000,C 90.000,E1 127.729} C_DIS
LIN {X -0.055,Y -416.091,Z 637.507,A 0.000,B 0.000,C 90.000,E1 127.317} C_DIS
LIN {X 0.076,Y -419.643,Z 637.506,A 0.000,B 0.000,C 90.000,E1 126.996} C_DIS
LIN {X 0.061,Y -425.517,Z 637.503,A 0.000,B 0.000,C 90.000,E1 126.583} C_DIS
LIN {X -0.031,Y -447.482,Z 637.496,A 0.000,B 0.000,C 90.000,E1 125.231} C_DIS
LIN {X -0.117,Y -458.843,Z 637.492,A 0.000,B 0.000,C 90.000,E1 124.532} C_DIS
LIN {X -0.057,Y -471.653,Z 637.487,A 0.000,B 0.000,C 90.000,E1 123.658} C_DIS
LIN {X -0.048,Y -477.865,Z 637.485,A 0.000,B 0.000,C 90.000,E1 123.214} C_DIS
LIN {X -0.081,Y -487.034,Z 637.481,A 0.000,B 0.000,C 90.000,E1 122.546} C_DIS
LIN {X 0.113,Y -494.372,Z 637.478,A 0.000,B 0.000,C 90.000,E1 121.957} C_DIS
LIN {X -0.220,Y -498.431,Z 637.476,A 0.000,B 0.000,C 90.000,E1 121.671} C_DIS
LIN {X -0.090,Y -507.257,Z 637.472,A 0.000,B 0.000,C 90.000,E1 120.924} C_DIS
LIN {X 0.022,Y -512.960,Z 637.469,A 0.000,B 0.000,C 90.000,E1 120.413} C_DIS
LIN {X -0.004,Y -521.287,Z 637.465,A 0.000,B 0.000,C 90.000,E1 119.667} C_DIS
LIN {X 0.153,Y -530.711,Z 637.460,A 0.000,B 0.000,C 90.000,E1 118.743} C_DIS
LIN {X 0.120,Y -536.840,Z 637.456,A 0.000,B 0.000,C 90.000,E1 118.103} C_DIS
LIN {X -0.120,Y -541.711,Z 637.453,A 0.000,B 0.000,C 90.000,E1 117.564} C_DIS
LIN {X -0.159,Y -546.210,Z 637.450,A 0.000,B 0.000,C 90.000,E1 117.001} C_DIS
LIN {X 0.081,Y -550.146,Z 637.447,A 0.000,B 0.000,C 90.000,E1 116.411} C_DIS
LIN {X -0.008,Y -554.505,Z 637.443,A 0.000,B 0.000,C 90.000,E1 115.720} C_DIS
LIN {X 0.016,Y -558.920,Z 637.438,A 0.000,B 0.000,C 90.000,E1 114.899} C_DIS
LIN {X -0.095,Y -562.961,Z 637.434,A 0.000,B 0.000,C 90.000,E1 114.079} C_DIS
LIN {X 0.028,Y -565.491,Z 637.431,A 0.000,B 0.000,C 90.000,E1 113.515} C_DIS
LIN {X 0.103,Y -570.076,Z 637.425,A 0.000,B 0.000,C 90.000,E1 112.408} C_DIS
LIN {X -0.076,Y -574.110,Z 637.419,A 0.000,B 0.000,C 90.000,E1 111.334} C_DIS
LIN {X -0.091,Y -575.962,Z 637.416,A 0.000,B 0.000,C 90.000,E1 110.791} C_DIS
LIN {X 0.291,Y -578.551,Z 637.411,A 0.000,B 0.000,C 90.000,E1 109.939} C_DIS
LIN {X 0.155,Y -580.898,Z 637.406,A 0.000,B 0.000,C 90.000,E1 109.141} C_DIS
LIN {X -0.149,Y -583.019,Z 637.402,A 0.000,B 0.000,C 90.000,E1 108.362} C_DIS
LIN {X 0.132,Y -584.911,Z 637.398,A 0.000,B 0.000,C 90.000,E1 107.528} C_DIS
LIN {X -0.197,Y -588.585,Z 637.389,A 0.000,B 0.000,C 90.000,E1 105.953} C_DIS
LIN {X -0.223,Y -592.417,Z 637.380,A 0.000,B 0.000,C 90.000,E1 104.356} C_DIS
LIN {X -0.016,Y -596.955,Z 637.369,A 0.000,B 0.000,C 90.000,E1 102.479} C_DIS
LIN {X 0.306,Y -601.407,Z 637.359,A 0.000,B 0.000,C 90.000,E1 100.602} C_DIS
LIN {X -0.024,Y -604.446,Z 637.352,A 0.000,B 0.000,C 90.000,E1 99.321} C_DIS
LIN {X -0.038,Y -606.814,Z 637.346,A 0.000,B 0.000,C 90.000,E1 98.276} C_DIS
LIN {X 0.223,Y -609.485,Z 637.339,A 0.000,B 0.000,C 90.000,E1 96.947} C_DIS
LIN {X 0.195,Y -611.458,Z 637.333,A 0.000,B 0.000,C 90.000,E1 95.910} C_DIS
LIN {X -0.139,Y -613.677,Z 637.326,A 0.000,B 0.000,C 90.000,E1 94.645} C_DIS
LIN {X 0.134,Y -615.667,Z 637.319,A 0.000,B 0.000,C 90.000,E1 93.326} C_DIS
LIN {X 0.144,Y -617.051,Z 637.313,A 0.000,B 0.000,C 90.000,E1 92.293} C_DIS
LIN {X 0.166,Y -618.276,Z 637.307,A 0.000,B 0.000,C 90.000,E1 91.260} C_DIS
LIN {X -0.114,Y -619.308,Z 637.300,A 0.000,B 0.000,C 90.000,E1 90.000} C_DIS
LIN {X -0.078,Y -620.003,Z 637.294,A 0.000,B 0.000,C 90.000,E1 88.969} C_DIS
LIN {X 0.261,Y -620.274,Z 637.290,A 0.000,B 0.000,C 90.000,E1 88.167} C_DIS
LIN {X -0.297,Y -620.414,Z 637.284,A 0.000,B 0.000,C 90.000,E1 87.192} C_DIS
LIN {X 0.128,Y -620.213,Z 637.277,A 0.000,B 0.000,C 90.000,E1 85.869} C_DIS
LIN {X 0.192,Y -619.824,Z 637.271,A 0.000,B 0.000,C 90.000,E1 84.837} C_DIS
LIN {X -0.012,Y -619.107,Z 637.264,A 0.000,B 0.000,C 90.000,E1 83.571} C_DIS
LIN {X 0.084,Y -618.410,Z 637.259,A 0.000,B 0.000,C 90.000,E1 82.534} C_DIS
LIN {X -0.116,Y -617.658,Z 637.254,A 0.000,B 0.000,C 90.000,E1 81.781} C_DIS
LIN {X 0.046,Y -616.373,Z 637.249,A 0.000,B 0.000,C 90.000,E1 80.735} C_DIS
LIN {X -0.049,Y -614.549,Z 637.241,A 0.000,B 0.000,C 90.000,E1 79.454} C_DIS
LIN {X -0.178,Y -612.455,Z 637.234,A 0.000,B 0.000,C 90.000,E1 78.173} C_DIS
LIN {X 0.029,Y -610.616,Z 637.229,A 0.000,B 0.000,C 90.000,E1 77.117} C_DIS
LIN {X -0.047,Y -608.163,Z 637.221,A 0.000,B 0.000,C 90.000,E1 75.825} C_DIS
LIN {X -0.020,Y -605.479,Z 637.214,A 0.000,B 0.000,C 90.000,E1 74.519} C_DIS
LIN {X 0.234,Y -603.105,Z 637.208,A 0.000,B 0.000,C 90.000,E1 73.449} C_DIS
LIN {X -0.229,Y -600.059,Z 637.201,A 0.000,B 0.000,C 90.000,E1 72.181} C_DIS
LIN {X 0.129,Y -597.328,Z 637.195,A 0.000,B 0.000,C 90.000,E1 71.094} C_DIS
LIN {X -0.118,Y -594.152,Z 637.189,A 0.000,B 0.000,C 90.000,E1 70.061} C_DIS
LIN {X 0.141,Y -590.621,Z 637.183,A 0.000,B 0.000,C 90.000,E1 68.975} C_DIS
LIN {X 0.346,Y -587.719,Z 637.179,A 0.000,B 0.000,C 90.000,E1 68.156} C_DIS
LIN {X 0.179,Y -583.420,Z 637.173,A 0.000,B 0.000,C 90.000,E1 67.102} C_DIS
LIN {X 0.090,Y -580.041,Z 637.168,A 0.000,B 0.000,C 90.000,E1 66.305} C_DIS
LIN {X -0.111,Y -573.802,Z 637.161,A 0.000,B 0.000,C 90.000,E1 64.973} C_DIS
LIN {X -0.158,Y -568.895,Z 637.156,A 0.000,B 0.000,C 90.000,E1 64.024} C_DIS
LIN {X -0.087,Y -564.956,Z 637.152,A 0.000,B 0.000,C 90.000,E1 63.332} C_DIS
LIN {X 0.297,Y -561.626,Z 637.149,A 0.000,B 0.000,C 90.000,E1 62.743} C_DIS
LIN {X -0.044,Y -555.792,Z 637.144,A 0.000,B 0.000,C 90.000,E1 61.948} C_DIS
LIN {X 0.122,Y -552.731,Z 637.142,A 0.000,B 0.000,C 90.000,E1 61.513} C_DIS
LIN {X 0.072,Y -544.097,Z 637.136,A 0.000,B 0.000,C 90.000,E1 60.539} C_DIS
LIN {X -0.049,Y -542.807,Z 637.136,A 0.000,B 0.000,C 90.000,E1 60.411} C_DIS
LIN {X 0.115,Y -538.533,Z 637.133,A 0.000,B 0.000,C 90.000,E1 59.999} C_DIS
LIN {X 0.058,Y -534.575,Z 637.132,A 0.000,B 0.000,C 90.000,E1 59.665} C_DIS
LIN {X -0.202,Y -529.870,Z 637.130,A 0.000,B 0.000,C 90.000,E1 59.331} C_DIS
LIN {X 0.086,Y -526.782,Z 637.128,A 0.000,B 0.000,C 90.000,E1 59.076} C_DIS
LIN {X 0.171,Y -521.873,Z 637.127,A 0.000,B 0.000,C 90.000,E1 58.742} C_DIS
LIN {X 0.327,Y -515.153,Z 637.124,A 0.000,B 0.000,C 90.000,E1 58.329} C_DIS
LIN {X -0.092,Y -506.741,Z 637.122,A 0.000,B 0.000,C 90.000,E1 57.916} C_DIS
LIN {X 0.113,Y -489.963,Z 637.117,A 0.000,B 0.000,C 90.000,E1 57.041} C_DIS
LIN {X 0.023,Y -476.714,Z 637.113,A 0.000,B 0.000,C 90.000,E1 56.373} C_DIS
LIN {X 0.260,Y -458.189,Z 637.108,A 0.000,B 0.000,C 90.000,E1 55.388} C_DIS
LIN {X 0.244,Y -441.511,Z 637.103,A 0.000,B 0.000,C 90.000,E1 54.482} C_DIS
LIN {X 0.018,Y -438.741,Z 637.102,A 0.000,B 0.000,C 90.000,E1 54.356} C_DIS
LIN {X -0.026,Y -438.674,Z 637.102,A 0.000,B 0.000,C 90.000,E1 54.356} C_DIS
LIN {X 0.008,Y -431.717,Z 637.083,A 0.000,B 0.000,C 90.000,E1 50.928} C_DIS
LIN {X -0.084,Y -430.113,Z 637.079,A 0.000,B 0.000,C 90.000,E1 50.275} C_DIS
LIN {X -0.050,Y -424.132,Z 637.065,A 0.000,B 0.000,C 90.000,E1 47.676} C_DIS
LIN {X 0.166,Y -424.613,Z 637.057,A 0.000,B 0.000,C 90.000,E1 46.215} C_DIS
LIN {X -0.206,Y -424.888,Z 637.049,A 0.000,B 0.000,C 90.000,E1 44.919} C_DIS
LIN {X -0.036,Y -425.453,Z 637.034,A 0.000,B 0.000,C 90.000,E1 42.204} C_DIS
LIN {X 0.209,Y -426.449,Z 637.020,A 0.000,B 0.000,C 90.000,E1 39.483} C_DIS
LIN {X -0.192,Y -427.338,Z 637.008,A 0.000,B 0.000,C 90.000,E1 37.523} C_DIS
LIN {X 0.004,Y -428.557,Z 636.995,A 0.000,B 0.000,C 90.000,E1 35.152} C_DIS
LIN {X -0.154,Y -429.378,Z 636.984,A 0.000,B 0.000,C 90.000,E1 33.166} C_DIS
LIN {X 0.077,Y -430.310,Z 636.971,A 0.000,B 0.000,C 90.000,E1 30.797} C_DIS
LIN {X -0.119,Y -430.980,Z 636.962,A 0.000,B 0.000,C 90.000,E1 29.155} C_DIS
LIN {X 0.277,Y -431.575,Z 636.955,A 0.000,B 0.000,C 90.000,E1 27.769} C_DIS
LIN {X 0.098,Y -432.734,Z 636.942,A 0.000,B 0.000,C 90.000,E1 25.463} C_DIS
LIN {X -0.021,Y -433.938,Z 636.929,A 0.000,B 0.000,C 90.000,E1 23.153} C_DIS
LIN {X 0.079,Y -435.001,Z 636.919,A 0.000,B 0.000,C 90.000,E1 21.482} C_DIS
LIN {X 0.191,Y -436.006,Z 636.910,A 0.000,B 0.000,C 90.000,E1 19.812} C_DIS
LIN {X -0.150,Y -437.127,Z 636.899,A 0.000,B 0.000,C 90.000,E1 17.873} C_DIS
LIN {X -0.057,Y -438.530,Z 636.886,A 0.000,B 0.000,C 90.000,E1 15.552} C_DIS
LIN {X 0.219,Y -440.346,Z 636.872,A 0.000,B 0.000,C 90.000,E1 12.883} C_DIS
LIN {X 0.094,Y -442.223,Z 636.859,A 0.000,B 0.000,C 90.000,E1 10.602} C_DIS
LIN {X 0.207,Y -444.963,Z 636.843,A 0.000,B 0.000,C 90.000,E1 7.644} C_DIS
LIN {X -0.185,Y -446.957,Z 636.832,A 0.000,B 0.000,C 90.000,E1 5.739} C_DIS
LIN {X 0.189,Y -449.941,Z 636.817,A 0.000,B 0.000,C 90.000,E1 3.094} C_DIS
LIN {X -0.197,Y -452.378,Z 636.807,A 0.000,B 0.000,C 90.000,E1 1.203} C_DIS
LIN {X -0.028,Y -456.141,Z 636.792,A 0.000,B 0.000,C 90.000,E1 358.511} C_DIS
LIN {X 0.211,Y -459.230,Z 636.781,A 0.000,B 0.000,C 90.000,E1 356.560} C_DIS
LIN {X 0.064,Y -462.435,Z 636.770,A 0.000,B 0.000,C 90.000,E1 354.666} C_DIS
LIN {X 0.075,Y -465.724,Z 636.760,A 0.000,B 0.000,C 90.000,E1 352.761} C_DIS
LIN {X 0.046,Y -469.588,Z 636.748,A 0.000,B 0.000,C 90.000,E1 350.557} C_DIS
LIN {X 0.170,Y -471.744,Z 636.741,A 0.000,B 0.000,C 90.000,E1 349.285} C_DIS
LIN {X 0.002,Y -475.508,Z 636.728,A 0.000,B 0.000,C 90.000,E1 347.117} C_DIS
LIN {X 0.040,Y -479.469,Z 636.716,A 0.000,B 0.000,C 90.000,E1 344.936} C_DIS
LIN {X -0.021,Y -483.520,Z 636.704,A 0.000,B 0.000,C 90.000,E1 342.779} C_DIS
LIN {X 0.156,Y -486.527,Z 636.696,A 0.000,B 0.000,C 90.000,E1 341.221} C_DIS
LIN {X 0.081,Y -489.531,Z 636.687,A 0.000,B 0.000,C 90.000,E1 339.699} C_DIS
LIN {X 0.279,Y -493.083,Z 636.677,A 0.000,B 0.000,C 90.000,E1 337.847} C_DIS
LIN {X -0.047,Y -494.681,Z 636.672,A 0.000,B 0.000,C 90.000,E1 336.975} C_DIS
LIN {X -0.253,Y -497.171,Z 636.664,A 0.000,B 0.000,C 90.000,E1 335.485} C_DIS
LIN {X 0.059,Y -499.967,Z 636.654,A 0.000,B 0.000,C 90.000,E1 333.640} C_DIS
LIN {X -0.016,Y -502.745,Z 636.644,A 0.000,B 0.000,C 90.000,E1 331.847} C_DIS
LIN {X 0.225,Y -508.481,Z 636.625,A 0.000,B 0.000,C 90.000,E1 328.535} C_DIS
LIN {X 0.079,Y -510.461,Z 636.620,A 0.000,B 0.000,C 90.000,E1 327.661} C_DIS
LIN {X 0.321,Y -512.287,Z 636.617,A 0.000,B 0.000,C 90.000,E1 327.041} C_DIS
LIN {X 0.049,Y -513.698,Z 636.615,A 0.000,B 0.000,C 90.000,E1 326.628} C_DIS
LIN {X -0.215,Y -515.471,Z 636.612,A 0.000,B 0.000,C 90.000,E1 326.215} C_DIS
LIN {X 0.137,Y -517.032,Z 636.611,A 0.000,B 0.000,C 90.000,E1 325.881} C_DIS
LIN {X -0.110,Y -519.960,Z 636.608,A 0.000,B 0.000,C 90.000,E1 325.468} C_DIS
LIN {X 0.108,Y -524.034,Z 636.606,A 0.000,B 0.000,C 90.000,E1 324.975} C_DIS
LIN {X 0.151,Y -532.651,Z 636.601,A 0.000,B 0.000,C 90.000,E1 324.196} C_DIS
LIN {X 0.327,Y -545.791,Z 636.595,A 0.000,B 0.000,C 90.000,E1 323.130} C_DIS
LIN {X -0.259,Y -554.209,Z 636.591,A 0.000,B 0.000,C 90.000,E1 322.477} C_DIS
LIN {X 0.051,Y -565.494,Z 636.586,A 0.000,B 0.000,C 90.000,E1 321.492} C_DIS
LIN {X -0.278,Y -573.816,Z 636.582,A 0.000,B 0.000,C 90.000,E1 320.803} C_DIS
LIN {X 0.189,Y -583.420,Z 636.577,A 0.000,B 0.000,C 90.000,E1 319.908} C_DIS
LIN {X 0.208,Y -590.103,Z 636.574,A 0.000,B 0.000,C 90.000,E1 319.299} C_DIS
LIN {X 0.159,Y -598.032,Z 636.570,A 0.000,B 0.000,C 90.000,E1 318.566} C_DIS
LIN {X -0.275,Y -601.876,Z 636.568,A 0.000,B 0.000,C 90.000,E1 318.243} C_DIS
LIN {X 0.219,Y -610.472,Z 636.563,A 0.000,B 0.000,C 90.000,E1 317.310} C_DIS
LIN {X 0.179,Y -614.831,Z 636.560,A 0.000,B 0.000,C 90.000,E1 316.824} C_DIS
LIN {X -0.325,Y -619.022,Z 636.558,A 0.000,B 0.000,C 90.000,E1 316.377} C_DIS
LIN {X 0.249,Y -623.207,Z 636.555,A 0.000,B 0.000,C 90.000,E1 315.810} C_DIS
LIN {X 0.229,Y -630.061,Z 636.550,A 0.000,B 0.000,C 90.000,E1 314.919} C_DIS
LIN {X 0.389,Y -634.676,Z 636.546,A 0.000,B 0.000,C 90.000,E1 314.271} C_DIS
LIN {X -0.298,Y -640.930,Z 636.541,A 0.000,B 0.000,C 90.000,E1 313.461} C_DIS
LIN {X -0.144,Y -647.853,Z 636.536,A 0.000,B 0.000,C 90.000,E1 312.447} C_DIS
LIN {X -0.278,Y -652.047,Z 636.532,A 0.000,B 0.000,C 90.000,E1 311.838} C_DIS
LIN {X 0.066,Y -656.843,Z 636.528,A 0.000,B 0.000,C 90.000,E1 311.067} C_DIS
LIN {X 0.027,Y -661.116,Z 636.524,A 0.000,B 0.000,C 90.000,E1 310.334} C_DIS
LIN {X 0.004,Y -664.403,Z 636.521,A 0.000,B 0.000,C 90.000,E1 309.725} C_DIS
LIN {X 0.003,Y -667.438,Z 636.517,A 0.000,B 0.000,C 90.000,E1 309.116} C_DIS
LIN {X 0.075,Y -669.669,Z 636.515,A 0.000,B 0.000,C 90.000,E1 308.624} C_DIS
LIN {X 0.158,Y -673.784,Z 636.509,A 0.000,B 0.000,C 90.000,E1 307.649} C_DIS
LIN {X -0.128,Y -677.329,Z 636.504,A 0.000,B 0.000,C 90.000,E1 306.710} C_DIS
LIN {X 0.177,Y -680.599,Z 636.499,A 0.000,B 0.000,C 90.000,E1 305.724} C_DIS
LIN {X 0.137,Y -683.686,Z 636.493,A 0.000,B 0.000,C 90.000,E1 304.771} C_DIS
LIN {X 0.160,Y -687.298,Z 636.487,A 0.000,B 0.000,C 90.000,E1 303.579} C_DIS
LIN {X 0.217,Y -690.011,Z 636.481,A 0.000,B 0.000,C 90.000,E1 302.625} C_DIS
LIN {X 0.308,Y -692.547,Z 636.476,A 0.000,B 0.000,C 90.000,E1 301.671} C_DIS
LIN {X -0.284,Y -695.637,Z 636.470,A 0.000,B 0.000,C 90.000,E1 300.541} C_DIS
LIN {X 0.120,Y -698.390,Z 636.463,A 0.000,B 0.000,C 90.000,E1 299.333} C_DIS
LIN {X -0.051,Y -700.375,Z 636.458,A 0.000,B 0.000,C 90.000,E1 298.409} C_DIS
LIN {X 0.091,Y -702.258,Z 636.453,A 0.000,B 0.000,C 90.000,E1 297.462} C_DIS
LIN {X 0.306,Y -703.426,Z 636.449,A 0.000,B 0.000,C 90.000,E1 296.744} C_DIS
LIN {X -0.071,Y -704.042,Z 636.446,A 0.000,B 0.000,C 90.000,E1 296.309} C_DIS
LIN {X 0.154,Y -704.351,Z 636.442,A 0.000,B 0.000,C 90.000,E1 295.591} C_DIS
LIN {X -0.212,Y -703.368,Z 636.440,A 0.000,B 0.000,C 90.000,E1 295.155} C_DIS
LIN {X 0.072,Y -702.770,Z 636.438,A 0.000,B 0.000,C 90.000,E1 294.899} C_DIS
LIN {X 0.214,Y -702.183,Z 636.438,A 0.000,B 0.000,C 90.000,E1 294.771} C_DIS
LIN {X -0.162,Y -698.766,Z 636.435,A 0.000,B 0.000,C 90.000,E1 294.335} C_DIS
LIN {X -0.027,Y -697.748,Z 636.435,A 0.000,B 0.000,C 90.000,E1 294.207} C_DIS
LIN {X 0.105,Y -696.218,Z 636.434,A 0.000,B 0.000,C 90.000,E1 294.079} C_DIS
LIN {X 0.235,Y -693.663,Z 636.433,A 0.000,B 0.000,C 90.000,E1 293.951} C_DIS
LIN {X -0.006,Y -689.592,Z 636.432,A 0.000,B 0.000,C 90.000,E1 293.823} C_DIS
LIN {X 0.140,Y -685.995,Z 636.432,A 0.000,B 0.000,C 90.000,E1 293.695} C_DIS
LIN {X 0.080,Y -681.578,Z 636.431,A 0.000,B 0.000,C 90.000,E1 293.590} C_DIS
LIN {X -0.350,Y -673.148,Z 636.431,A 0.000,B 0.000,C 90.000,E1 293.515} C_DIS
LIN {X 0.404,Y -666.143,Z 636.430,A 0.000,B 0.000,C 90.000,E1 293.387} C_DIS
LIN {X -0.166,Y -649.901,Z 636.429,A 0.000,B 0.000,C 90.000,E1 293.206} C_DIS
LIN {X -0.081,Y -639.912,Z 636.428,A 0.000,B 0.000,C 90.000,E1 293.025} C_DIS
LIN {X -0.175,Y -630.228,Z 636.427,A 0.000,B 0.000,C 90.000,E1 292.823} C_DIS
LIN {X 0.007,Y -616.910,Z 636.425,A 0.000,B 0.000,C 90.000,E1 292.461} C_DIS
LIN {X -0.138,Y -599.956,Z 636.422,A 0.000,B 0.000,C 90.000,E1 291.972} C_DIS
LIN {X 0.024,Y -582.469,Z 636.419,A 0.000,B 0.000,C 90.000,E1 291.408} C_DIS
LIN {X 0.190,Y -575.267,Z 636.418,A 0.000,B 0.000,C 90.000,E1 291.173} C_DIS
LIN {X -0.209,Y -565.199,Z 636.416,A 0.000,B 0.000,C 90.000,E1 290.918} C_DIS
LIN {X -0.186,Y -560.875,Z 636.415,A 0.000,B 0.000,C 90.000,E1 290.737} C_DIS
LIN {X -0.189,Y -559.322,Z 636.415,A 0.000,B 0.000,C 90.000,E1 290.663} C_DIS
LIN {X 0.226,Y -556.829,Z 636.414,A 0.000,B 0.000,C 90.000,E1 290.429} C_DIS
LIN {X 0.192,Y -556.797,Z 636.414,A 0.000,B 0.000,C 90.000,E1 290.429} C_DIS
LIN {X -0.111,Y -555.960,Z 636.412,A 0.000,B 0.000,C 90.000,E1 290.248} C_DIS
LIN {X 0.064,Y -555.652,Z 636.410,A 0.000,B 0.000,C 90.000,E1 289.812} C_DIS
LIN {X 0.221,Y -555.776,Z 636.406,A 0.000,B 0.000,C 90.000,E1 288.960} C_DIS
LIN {X -0.043,Y -555.704,Z 636.399,A 0.000,B 0.000,C 90.000,E1 287.873} C_DIS
LIN {X 0.220,Y -555.462,Z 636.393,A 0.000,B 0.000,C 90.000,E1 286.732} C_DIS
LIN {X -0.211,Y -555.123,Z 636.387,A 0.000,B 0.000,C 90.000,E1 285.662} C_DIS
LIN {X 0.016,Y -554.519,Z 636.379,A 0.000,B 0.000,C 90.000,E1 284.245} C_DIS
LIN {X -0.182,Y -553.658,Z 636.370,A 0.000,B 0.000,C 90.000,E1 282.591} C_DIS
LIN {X 0.139,Y -552.648,Z 636.359,A 0.000,B 0.000,C 90.000,E1 280.602} C_DIS
LIN {X -0.217,Y -551.879,Z 636.348,A 0.000,B 0.000,C 90.000,E1 278.681} C_DIS
LIN {X 0.297,Y -551.189,Z 636.339,A 0.000,B 0.000,C 90.000,E1 276.947} C_DIS
LIN {X 0.235,Y -550.585,Z 636.328,A 0.000,B 0.000,C 90.000,E1 274.992} C_DIS
LIN {X 0.074,Y -550.129,Z 636.319,A 0.000,B 0.000,C 90.000,E1 273.326} C_DIS
LIN {X -0.178,Y -549.772,Z 636.311,A 0.000,B 0.000,C 90.000,E1 271.949} C_DIS
LIN {X 0.162,Y -549.252,Z 636.301,A 0.000,B 0.000,C 90.000,E1 270.229} C_DIS
LIN {X -0.124,Y -548.619,Z 636.294,A 0.000,B 0.000,C 90.000,E1 268.854} C_DIS
LIN {X 0.139,Y -547.955,Z 636.286,A 0.000,B 0.000,C 90.000,E1 267.421} C_DIS
LIN {X -0.202,Y -547.421,Z 636.280,A 0.000,B 0.000,C 90.000,E1 266.331} C_DIS
LIN {X 0.037,Y -546.774,Z 636.273,A 0.000,B 0.000,C 90.000,E1 265.179} C_DIS
LIN {X 0.188,Y -546.162,Z 636.269,A 0.000,B 0.000,C 90.000,E1 264.318} C_DIS
LIN {X -0.048,Y -545.150,Z 636.261,A 0.000,B 0.000,C 90.000,E1 262.932} C_DIS
LIN {X 0.143,Y -544.293,Z 636.256,A 0.000,B 0.000,C 90.000,E1 262.064} C_DIS
LIN {X -0.132,Y -542.765,Z 636.248,A 0.000,B 0.000,C 90.000,E1 260.679} C_DIS
LIN {X -0.051,Y -540.314,Z 636.234,A 0.000,B 0.000,C 90.000,E1 258.117} C_DIS
LIN {X 0.100,Y -538.411,Z 636.221,A 0.000,B 0.000,C 90.000,E1 255.825} C_DIS
LIN {X -0.042,Y -537.436,Z 636.215,A 0.000,B 0.000,C 90.000,E1 254.700} C_DIS
LIN {X 0.199,Y -535.644,Z 636.206,A 0.000,B 0.000,C 90.000,E1 252.960} C_DIS
LIN {X -0.101,Y -533.987,Z 636.196,A 0.000,B 0.000,C 90.000,E1 251.275} C_DIS
LIN {X -0.178,Y -533.089,Z 636.191,A 0.000,B 0.000,C 90.000,E1 250.423} C_DIS
LIN {X -0.068,Y -531.532,Z 636.185,A 0.000,B 0.000,C 90.000,E1 249.263} C_DIS
LIN {X 0.203,Y -529.460,Z 636.177,A 0.000,B 0.000,C 90.000,E1 247.794} C_DIS
LIN {X 0.141,Y -527.135,Z 636.169,A 0.000,B 0.000,C 90.000,E1 246.357} C_DIS
LIN {X 0.181,Y -525.561,Z 636.164,A 0.000,B 0.000,C 90.000,E1 245.485} C_DIS
LIN {X 0.108,Y -523.231,Z 636.158,A 0.000,B 0.000,C 90.000,E1 244.332} C_DIS
LIN {X -0.174,Y -519.502,Z 636.148,A 0.000,B 0.000,C 90.000,E1 242.615} C_DIS
LIN {X 0.029,Y -516.399,Z 636.140,A 0.000,B 0.000,C 90.000,E1 241.129} C_DIS
LIN {X 0.064,Y -513.763,Z 636.133,A 0.000,B 0.000,C 90.000,E1 239.950} C_DIS
LIN {X 0.222,Y -510.260,Z 636.125,A 0.000,B 0.000,C 90.000,E1 238.456} C_DIS
LIN {X -0.001,Y -507.448,Z 636.118,A 0.000,B 0.000,C 90.000,E1 237.296} C_DIS
LIN {X 0.049,Y -503.761,Z 636.110,A 0.000,B 0.000,C 90.000,E1 235.801} C_DIS
LIN {X 0.129,Y -501.463,Z 636.105,A 0.000,B 0.000,C 90.000,E1 234.895} C_DIS
LIN {X -0.071,Y -497.550,Z 636.097,A 0.000,B 0.000,C 90.000,E1 233.417} C_DIS
LIN {X -0.175,Y -491.435,Z 636.083,A 0.000,B 0.000,C 90.000,E1 231.009} C_DIS
LIN {X -0.130,Y -486.923,Z 636.073,A 0.000,B 0.000,C 90.000,E1 229.175} C_DIS
LIN {X -0.061,Y -483.196,Z 636.065,A 0.000,B 0.000,C 90.000,E1 227.634} C_DIS
LIN {X 0.267,Y -479.516,Z 636.056,A 0.000,B 0.000,C 90.000,E1 226.053} C_DIS
LIN {X -0.276,Y -474.246,Z 636.044,A 0.000,B 0.000,C 90.000,E1 223.947} C_DIS
LIN {X -0.121,Y -470.681,Z 636.035,A 0.000,B 0.000,C 90.000,E1 222.366} C_DIS
LIN {X 0.067,Y -466.566,Z 636.025,A 0.000,B 0.000,C 90.000,E1 220.458} C_DIS
LIN {X 0.056,Y -463.853,Z 636.018,A 0.000,B 0.000,C 90.000,E1 219.197} C_DIS
LIN {X -0.120,Y -459.202,Z 636.005,A 0.000,B 0.000,C 90.000,E1 216.996} C_DIS
LIN {X 0.034,Y -454.864,Z 635.993,A 0.000,B 0.000,C 90.000,E1 214.739} C_DIS
LIN {X 0.047,Y -452.485,Z 635.986,A 0.000,B 0.000,C 90.000,E1 213.452} C_DIS
LIN {X -0.180,Y -448.992,Z 635.975,A 0.000,B 0.000,C 90.000,E1 211.544} C_DIS
LIN {X 0.131,Y -446.682,Z 635.968,A 0.000,B 0.000,C 90.000,E1 210.207} C_DIS
LIN {X -0.207,Y -444.447,Z 635.961,A 0.000,B 0.000,C 90.000,E1 208.949} C_DIS
LIN {X 0.132,Y -440.351,Z 635.948,A 0.000,B 0.000,C 90.000,E1 206.616} C_DIS
LIN {X 0.109,Y -437.368,Z 635.939,A 0.000,B 0.000,C 90.000,E1 204.975} C_DIS
LIN {X -0.146,Y -433.230,Z 635.926,A 0.000,B 0.000,C 90.000,E1 202.695} C_DIS
LIN {X -0.066,Y -429.159,Z 635.913,A 0.000,B 0.000,C 90.000,E1 200.355} C_DIS
LIN {X 0.021,Y -426.322,Z 635.904,A 0.000,B 0.000,C 90.000,E1 198.671} C_DIS
LIN {X -0.156,Y -423.116,Z 635.893,A 0.000,B 0.000,C 90.000,E1 196.677} C_DIS
LIN {X 0.102,Y -420.480,Z 635.883,A 0.000,B 0.000,C 90.000,E1 194.954} C_DIS
LIN {X 0.143,Y -418.400,Z 635.876,A 0.000,B 0.000,C 90.000,E1 193.592} C_DIS
LIN {X -0.114,Y -414.737,Z 635.862,A 0.000,B 0.000,C 90.000,E1 191.243} C_DIS
LIN {X 0.183,Y -411.316,Z 635.849,A 0.000,B 0.000,C 90.000,E1 188.803} C_DIS
LIN {X -0.087,Y -407.830,Z 635.836,A 0.000,B 0.000,C 90.000,E1 186.429} C_DIS
LIN {X -0.179,Y -404.251,Z 635.820,A 0.000,B 0.000,C 90.000,E1 183.669} C_DIS
LIN {X 0.052,Y -401.884,Z 635.809,A 0.000,B 0.000,C 90.000,E1 181.547} C_DIS
LIN {X 0.022,Y -398.738,Z 635.789,A 0.000,B 0.000,C 90.000,E1 178.051} C_DIS
LIN {X 0.160,Y -396.325,Z 635.764,A 0.000,B 0.000,C 90.000,E1 173.457} C_DIS
LIN {X -0.077,Y -395.745,Z 635.752,A 0.000,B 0.000,C 90.000,E1 171.376} C_DIS
LIN {X 0.132,Y -395.349,Z 635.736,A 0.000,B 0.000,C 90.000,E1 168.522} C_DIS
LIN {X 0.052,Y -395.401,Z 635.723,A 0.000,B 0.000,C 90.000,E1 166.061} C_DIS
LIN {X -0.101,Y -395.800,Z 635.705,A 0.000,B 0.000,C 90.000,E1 162.906} C_DIS
LIN {X -0.080,Y -396.169,Z 635.693,A 0.000,B 0.000,C 90.000,E1 160.786} C_DIS
LIN {X -0.186,Y -396.498,Z 635.685,A 0.000,B 0.000,C 90.000,E1 159.390} C_DIS
LIN {X -0.084,Y -396.957,Z 635.676,A 0.000,B 0.000,C 90.000,E1 157.614} C_DIS
LIN {X 0.027,Y -397.492,Z 635.664,A 0.000,B 0.000,C 90.000,E1 155.485} C_DIS
LIN {X -0.039,Y -398.134,Z 635.652,A 0.000,B 0.000,C 90.000,E1 153.384} C_DIS
LIN {X 0.087,Y -398.702,Z 635.640,A 0.000,B 0.000,C 90.000,E1 151.257} C_DIS
LIN {X -0.164,Y -399.211,Z 635.631,A 0.000,B 0.000,C 90.000,E1 149.537} C_DIS
LIN {X -0.198,Y -399.698,Z 635.621,A 0.000,B 0.000,C 90.000,E1 147.788} C_DIS
LIN {X -0.006,Y -400.306,Z 635.611,A 0.000,B 0.000,C 90.000,E1 146.008} C_DIS
LIN {X 0.097,Y -401.279,Z 635.598,A 0.000,B 0.000,C 90.000,E1 143.543} C_DIS
LIN {X -0.105,Y -401.992,Z 635.588,A 0.000,B 0.000,C 90.000,E1 141.823} C_DIS
LIN {X -0.050,Y -402.681,Z 635.578,A 0.000,B 0.000,C 90.000,E1 140.070} C_DIS
LIN {X -0.160,Y -403.168,Z 635.570,A 0.000,B 0.000,C 90.000,E1 138.690} C_DIS
LIN {X 0.090,Y -404.044,Z 635.557,A 0.000,B 0.000,C 90.000,E1 136.215} C_DIS
LIN {X -0.181,Y -404.698,Z 635.547,A 0.000,B 0.000,C 90.000,E1 134.514} C_DIS
LIN {X 0.046,Y -407.128,Z 635.522,A 0.000,B 0.000,C 90.000,E1 129.967} C_DIS
LIN {X 0.172,Y -408.331,Z 635.516,A 0.000,B 0.000,C 90.000,E1 128.910} C_DIS
LIN {X 0.004,Y -409.197,Z 635.514,A 0.000,B 0.000,C 90.000,E1 128.588} C_DIS
LIN {X -0.183,Y -410.265,Z 635.512,A 0.000,B 0.000,C 90.000,E1 128.096} C_DIS
LIN {X -0.026,Y -411.758,Z 635.510,A 0.000,B 0.000,C 90.000,E1 127.729} C_DIS
LIN {X -0.092,Y -412.619,Z 635.508,A 0.000,B 0.000,C 90.000,E1 127.523} C_DIS
LIN {X -0.196,Y -414.879,Z 635.507,A 0.000,B 0.000,C 90.000,E1 127.237} C_DIS
LIN {X -0.022,Y -418.455,Z 635.505,A 0.000,B 0.000,C 90.000,E1 126.870} C_DIS
LIN {X 0.120,Y -423.876,Z 635.503,A 0.000,B 0.000,C 90.000,E1 126.457} C_DIS
LIN {X 0.074,Y -448.608,Z 635.494,A 0.000,B 0.000,C 90.000,E1 124.945} C_DIS
LIN {X 0.213,Y -458.394,Z 635.491,A 0.000,B 0.000,C 90.000,E1 124.326} C_DIS
LIN {X 0.034,Y -471.121,Z 635.486,A 0.000,B 0.000,C 90.000,E1 123.499} C_DIS
LIN {X -0.169,Y -477.379,Z 635.484,A 0.000,B 0.000,C 90.000,E1 123.086} C_DIS
LIN {X -0.264,Y -486.749,Z 635.480,A 0.000,B 0.000,C 90.000,E1 122.418} C_DIS
LIN {X 0.132,Y -496.010,Z 635.476,A 0.000,B 0.000,C 90.000,E1 121.671} C_DIS
LIN {X -0.042,Y -506.321,Z 635.471,A 0.000,B 0.000,C 90.000,E1 120.846} C_DIS
LIN {X 0.107,Y -513.496,Z 635.468,A 0.000,B 0.000,C 90.000,E1 120.207} C_DIS
LIN {X -0.054,Y -522.048,Z 635.464,A 0.000,B 0.000,C 90.000,E1 119.461} C_DIS
LIN {X -0.269,Y -530.344,Z 635.459,A 0.000,B 0.000,C 90.000,E1 118.693} C_DIS
LIN {X -0.094,Y -535.408,Z 635.456,A 0.000,B 0.000,C 90.000,E1 118.153} C_DIS
LIN {X -0.192,Y -540.096,Z 635.453,A 0.000,B 0.000,C 90.000,E1 117.641} C_DIS
LIN {X -0.226,Y -544.376,Z 635.451,A 0.000,B 0.000,C 90.000,E1 117.129} C_DIS
LIN {X -0.066,Y -546.240,Z 635.449,A 0.000,B 0.000,C 90.000,E1 116.873} C_DIS
LIN {X 0.170,Y -548.218,Z 635.448,A 0.000,B 0.000,C 90.000,E1 116.565} C_DIS
LIN {X -0.050,Y -549.989,Z 635.446,A 0.000,B 0.000,C 90.000,E1 116.360} C_DIS
LIN {X 0.014,Y -554.339,Z 635.443,A 0.000,B 0.000,C 90.000,E1 115.668} C_DIS
LIN {X -0.320,Y -556.640,Z 635.440,A 0.000,B 0.000,C 90.000,E1 115.283} C_DIS
LIN {X -0.338,Y -558.164,Z 635.439,A 0.000,B 0.000,C 90.000,E1 115.027} C_DIS
LIN {X -0.045,Y -562.986,Z 635.434,A 0.000,B 0.000,C 90.000,E1 114.027} C_DIS
LIN {X -0.015,Y -566.163,Z 635.430,A 0.000,B 0.000,C 90.000,E1 113.334} C_DIS
LIN {X -0.056,Y -569.641,Z 635.425,A 0.000,B 0.000,C 90.000,E1 112.514} C_DIS
LIN {X -0.283,Y -572.815,Z 635.421,A 0.000,B 0.000,C 90.000,E1 111.716} C_DIS
LIN {X 0.062,Y -575.739,Z 635.416,A 0.000,B 0.000,C 90.000,E1 110.865} C_DIS
LIN {X -0.097,Y -578.416,Z 635.411,A 0.000,B 0.000,C 90.000,E1 110.066} C_DIS
LIN {X -0.234,Y -580.845,Z 635.407,A 0.000,B 0.000,C 90.000,E1 109.268} C_DIS
LIN {X 0.201,Y -583.016,Z 635.402,A 0.000,B 0.000,C 90.000,E1 108.417} C_DIS
LIN {X -0.078,Y -584.978,Z 635.398,A 0.000,B 0.000,C 90.000,E1 107.638} C_DIS
LIN {X -0.013,Y -588.679,Z 635.389,A 0.000,B 0.000,C 90.000,E1 106.024} C_DIS
LIN {X -0.024,Y -592.558,Z 635.380,A 0.000,B 0.000,C 90.000,E1 104.426} C_DIS
LIN {X -0.250,Y -597.163,Z 635.370,A 0.000,B 0.000,C 90.000,E1 102.591} C_DIS
LIN {X 0.068,Y -601.681,Z 635.360,A 0.000,B 0.000,C 90.000,E1 100.715} C_DIS
LIN {X 0.332,Y -604.776,Z 635.352,A 0.000,B 0.000,C 90.000,E1 99.378} C_DIS
LIN {X -0.041,Y -607.734,Z 635.345,A 0.000,B 0.000,C 90.000,E1 98.106} C_DIS
LIN {X 0.243,Y -610.430,Z 635.338,A 0.000,B 0.000,C 90.000,E1 96.777} C_DIS
LIN {X 0.231,Y -612.417,Z 635.332,A 0.000,B 0.000,C 90.000,E1 95.739} C_DIS
LIN {X 0.242,Y -614.188,Z 635.326,A 0.000,B 0.000,C 90.000,E1 94.702} C_DIS
LIN {X -0.091,Y -616.241,Z 635.319,A 0.000,B 0.000,C 90.000,E1 93.440} C_DIS
LIN {X -0.075,Y -617.663,Z 635.313,A 0.000,B 0.000,C 90.000,E1 92.407} C_DIS
LIN {X 0.269,Y -619.145,Z 635.306,A 0.000,B 0.000,C 90.000,E1 91.088} C_DIS
LIN {X 0.005,Y -620.172,Z 635.299,A 0.000,B 0.000,C 90.000,E1 89.828} C_DIS
LIN {X 0.053,Y -620.784,Z 635.293,A 0.000,B 0.000,C 90.000,E1 88.797} C_DIS
LIN {X -0.200,Y -621.024,Z 635.289,A 0.000,B 0.000,C 90.000,E1 88.051} C_DIS
LIN {X 0.149,Y -621.144,Z 635.285,A 0.000,B 0.000,C 90.000,E1 87.249} C_DIS
LIN {X -0.077,Y -620.938,Z 635.278,A 0.000,B 0.000,C 90.000,E1 85.988} C_DIS
LIN {X 0.042,Y -620.565,Z 635.272,A 0.000,B 0.000,C 90.000,E1 84.951} C_DIS
LIN {X -0.147,Y -619.834,Z 635.265,A 0.000,B 0.000,C 90.000,E1 83.685} C_DIS
LIN {X -0.037,Y -619.119,Z 635.259,A 0.000,B 0.000,C 90.000,E1 82.648} C_DIS
LIN {X -0.228,Y -618.357,Z 635.255,A 0.000,B 0.000,C 90.000,E1 81.894} C_DIS
LIN {X -0.053,Y -617.092,Z 635.249,A 0.000,B 0.000,C 90.000,E1 80.849} C_DIS
LIN {X -0.131,Y -615.243,Z 635.242,A 0.000,B 0.000,C 90.000,E1 79.567} C_DIS
LIN {X -0.243,Y -613.124,Z 635.235,A 0.000,B 0.000,C 90.000,E1 78.285} C_DIS
LIN {X -0.022,Y -611.289,Z 635.229,A 0.000,B 0.000,C 90.000,E1 77.229} C_DIS
LIN {X -0.081,Y -608.784,Z 635.222,A 0.000,B 0.000,C 90.000,E1 75.936} C_DIS
LIN {X -0.035,Y -606.062,Z 635.215,A 0.000,B 0.000,C 90.000,E1 74.629} C_DIS
LIN {X 0.232,Y -603.674,Z 635.209,A 0.000,B 0.000,C 90.000,E1 73.559} C_DIS
LIN {X 0.176,Y -600.565,Z 635.202,A 0.000,B 0.000,C 90.000,E1 72.253} C_DIS
LIN {X 0.257,Y -598.557,Z 635.197,A 0.000,B 0.000,C 90.000,E1 71.456} C_DIS
LIN {X 0.130,Y -596.259,Z 635.193,A 0.000,B 0.000,C 90.000,E1 70.678} C_DIS
LIN {X 0.176,Y -593.745,Z 635.188,A 0.000,B 0.000,C 90.000,E1 69.880} C_DIS
LIN {X -0.125,Y -590.038,Z 635.182,A 0.000,B 0.000,C 90.000,E1 68.847} C_DIS
LIN {X 0.195,Y -588.080,Z 635.180,A 0.000,B 0.000,C 90.000,E1 68.284} C_DIS
LIN {X 0.031,Y -583.732,Z 635.174,A 0.000,B 0.000,C 90.000,E1 67.230} C_DIS
LIN {X -0.123,Y -579.681,Z 635.168,A 0.000,B 0.000,C 90.000,E1 66.305} C_DIS
LIN {X -0.252,Y -573.960,Z 635.162,A 0.000,B 0.000,C 90.000,E1 65.101} C_DIS
LIN {X 0.029,Y -571.866,Z 635.159,A 0.000,B 0.000,C 90.000,E1 64.665} C_DIS
LIN {X -0.299,Y -568.998,Z 635.156,A 0.000,B 0.000,C 90.000,E1 64.152} C_DIS
LIN {X 0.026,Y -565.031,Z 635.152,A 0.000,B 0.000,C 90.000,E1 63.435} C_DIS
LIN {X -0.156,Y -563.156,Z 635.151,A 0.000,B 0.000,C 90.000,E1 63.179} C_DIS
LIN {X -0.004,Y -560.931,Z 635.149,A 0.000,B 0.000,C 90.000,E1 62.794} C_DIS
LIN {X -0.009,Y -555.939,Z 635.145,A 0.000,B 0.000,C 90.000,E1 62.103} C_DIS
LIN {X -0.177,Y -551.714,Z 635.142,A 0.000,B 0.000,C 90.000,E1 61.563} C_DIS
LIN {X -0.142,Y -546.641,Z 635.139,A 0.000,B 0.000,C 90.000,E1 61.001} C_DIS
LIN {X -0.175,Y -542.895,Z 635.137,A 0.000,B 0.000,C 90.000,E1 60.589} C_DIS
LIN {X -0.025,Y -537.171,Z 635.134,A 0.000,B 0.000,C 90.000,E1 60.049} C_DIS
LIN {X 0.276,Y -531.087,Z 635.131,A 0.000,B 0.000,C 90.000,E1 59.537} C_DIS
LIN {X 0.243,Y -526.412,Z 635.129,A 0.000,B 0.000,C 90.000,E1 59.203} C_DIS
LIN {X 0.117,Y -519.684,Z 635.127,A 0.000,B 0.000,C 90.000,E1 58.791} C_DIS
LIN {X 0.130,Y -512.898,Z 635.125,A 0.000,B 0.000,C 90.000,E1 58.408} C_DIS
LIN {X -0.094,Y -506.119,Z 635.123,A 0.000,B 0.000,C 90.000,E1 58.074} C_DIS
LIN {X -0.209,Y -491.199,Z 635.118,A 0.000,B 0.000,C 90.000,E1 57.327} C_DIS
LIN {X -0.038,Y -472.836,Z 635.113,A 0.000,B 0.000,C 90.000,E1 56.373} C_DIS
LIN {X -0.128,Y -446.071,Z 635.105,A 0.000,B 0.000,C 90.000,E1 54.975} C_DIS
LIN {X -0.166,Y -439.268,Z 635.103,A 0.000,B 0.000,C 90.000,E1 54.609} C_DIS
LIN {X 0.150,Y -439.206,Z 635.103,A 0.000,B 0.000,C 90.000,E1 54.562} C_DIS
LIN {X -0.157,Y -431.439,Z 635.082,A 0.000,B 0.000,C 90.000,E1 50.803} C_DIS
LIN {X 0.140,Y -424.544,Z 635.066,A 0.000,B 0.000,C 90.000,E1 47.838} C_DIS
LIN {X 0.056,Y -425.087,Z 635.058,A 0.000,B 0.000,C 90.000,E1 46.419} C_DIS
LIN {X -0.001,Y -425.387,Z 635.050,A 0.000,B 0.000,C 90.000,E1 45.081} C_DIS
LIN {X -0.034,Y -425.900,Z 635.037,A 0.000,B 0.000,C 90.000,E1 42.732} C_DIS
LIN {X -0.010,Y -426.715,Z 635.024,A 0.000,B 0.000,C 90.000,E1 40.378} C_DIS
LIN {X -0.141,Y -427.582,Z 635.013,A 0.000,B 0.000,C 90.000,E1 38.382} C_DIS
LIN {X -0.174,Y -428.516,Z 635.002,A 0.000,B 0.000,C 90.000,E1 36.377} C_DIS
LIN {X -0.070,Y -429.210,Z 634.995,A 0.000,B 0.000,C 90.000,E1 35.025} C_DIS
LIN {X -0.204,Y -429.743,Z 634.987,A 0.000,B 0.000,C 90.000,E1 33.706} C_DIS
LIN {X 0.027,Y -430.136,Z 634.982,A 0.000,B 0.000,C 90.000,E1 32.673} C_DIS
LIN {X 0.041,Y -430.791,Z 634.972,A 0.000,B 0.000,C 90.000,E1 31.003} C_DIS
LIN {X 0.069,Y -431.454,Z 634.963,A 0.000,B 0.000,C 90.000,E1 29.333} C_DIS
LIN {X 0.271,Y -432.181,Z 634.954,A 0.000,B 0.000,C 90.000,E1 27.641} C_DIS
LIN {X 0.107,Y -433.312,Z 634.941,A 0.000,B 0.000,C 90.000,E1 25.335} C_DIS
LIN {X 0.003,Y -434.474,Z 634.928,A 0.000,B 0.000,C 90.000,E1 23.025} C_DIS
LIN {X -0.123,Y -435.306,Z 634.921,A 0.000,B 0.000,C 90.000,E1 21.716} C_DIS
LIN {X -0.159,Y -436.284,Z 634.911,A 0.000,B 0.000,C 90.000,E1 20.066} C_DIS
LIN {X 0.064,Y -437.365,Z 634.900,A 0.000,B 0.000,C 90.000,E1 18.055} C_DIS
LIN {X -0.257,Y -438.758,Z 634.888,A 0.000,B 0.000,C 90.000,E1 15.788} C_DIS
LIN {X 0.024,Y -440.507,Z 634.873,A 0.000,B 0.000,C 90.000,E1 13.119} C_DIS
LIN {X -0.096,Y -442.342,Z 634.860,A 0.000,B 0.000,C 90.000,E1 10.838} C_DIS
LIN {X 0.201,Y -445.335,Z 634.842,A 0.000,B 0.000,C 90.000,E1 7.530} C_DIS
LIN {X -0.181,Y -447.304,Z 634.831,A 0.000,B 0.000,C 90.000,E1 5.625} C_DIS
LIN {X 0.030,Y -449.872,Z 634.819,A 0.000,B 0.000,C 90.000,E1 3.326} C_DIS
LIN {X -0.045,Y -451.876,Z 634.810,A 0.000,B 0.000,C 90.000,E1 1.718} C_DIS
LIN {X -0.206,Y -455.850,Z 634.794,A 0.000,B 0.000,C 90.000,E1 358.854} C_DIS
LIN {X 0.217,Y -459.353,Z 634.781,A 0.000,B 0.000,C 90.000,E1 356.560} C_DIS
LIN {X -0.146,Y -463.107,Z 634.769,A 0.000,B 0.000,C 90.000,E1 354.375} C_DIS
LIN {X -0.114,Y -466.348,Z 634.758,A 0.000,B 0.000,C 90.000,E1 352.470} C_DIS
LIN {X 0.060,Y -469.709,Z 634.748,A 0.000,B 0.000,C 90.000,E1 350.557} C_DIS
LIN {X 0.010,Y -472.352,Z 634.739,A 0.000,B 0.000,C 90.000,E1 348.993} C_DIS
LIN {X 0.020,Y -475.599,Z 634.729,A 0.000,B 0.000,C 90.000,E1 347.117} C_DIS
LIN {X 0.062,Y -479.534,Z 634.716,A 0.000,B 0.000,C 90.000,E1 344.936} C_DIS
LIN {X 0.001,Y -483.563,Z 634.704,A 0.000,B 0.000,C 90.000,E1 342.779} C_DIS
LIN {X -0.290,Y -485.975,Z 634.698,A 0.000,B 0.000,C 90.000,E1 341.583} C_DIS
LIN {X 0.083,Y -489.012,Z 634.689,A 0.000,B 0.000,C 90.000,E1 340.007} C_DIS
LIN {X 0.228,Y -491.938,Z 634.681,A 0.000,B 0.000,C 90.000,E1 338.465} C_DIS
LIN {X -0.110,Y -493.649,Z 634.675,A 0.000,B 0.000,C 90.000,E1 337.592} C_DIS
LIN {X 0.075,Y -495.689,Z 634.669,A 0.000,B 0.000,C 90.000,E1 336.357} C_DIS
LIN {X -0.227,Y -497.198,Z 634.664,A 0.000,B 0.000,C 90.000,E1 335.485} C_DIS
LIN {X 0.029,Y -499.512,Z 634.655,A 0.000,B 0.000,C 90.000,E1 333.948} C_DIS
LIN {X 0.013,Y -502.740,Z 634.644,A 0.000,B 0.000,C 90.000,E1 331.847} C_DIS
LIN {X -0.073,Y -507.776,Z 634.627,A 0.000,B 0.000,C 90.000,E1 328.869} C_DIS
LIN {X 0.006,Y -510.928,Z 634.619,A 0.000,B 0.000,C 90.000,E1 327.375} C_DIS
LIN {X -0.087,Y -511.904,Z 634.617,A 0.000,B 0.000,C 90.000,E1 327.089} C_DIS
LIN {X 0.070,Y -513.137,Z 634.615,A 0.000,B 0.000,C 90.000,E1 326.628} C_DIS
LIN {X -0.258,Y -515.634,Z 634.611,A 0.000,B 0.000,C 90.000,E1 326.008} C_DIS
LIN {X -0.071,Y -517.253,Z 634.609,A 0.000,B 0.000,C 90.000,E1 325.674} C_DIS
LIN {X 0.041,Y -517.891,Z 634.609,A 0.000,B 0.000,C 90.000,E1 325.515} C_DIS
LIN {X -0.105,Y -521.071,Z 634.606,A 0.000,B 0.000,C 90.000,E1 325.055} C_DIS
LIN {X 0.152,Y -524.041,Z 634.604,A 0.000,B 0.000,C 90.000,E1 324.689} C_DIS
LIN {X -0.277,Y -529.721,Z 634.601,A 0.000,B 0.000,C 90.000,E1 324.196} C_DIS
LIN {X -0.119,Y -536.866,Z 634.598,A 0.000,B 0.000,C 90.000,E1 323.577} C_DIS
LIN {X -0.130,Y -544.141,Z 634.594,A 0.000,B 0.000,C 90.000,E1 323.004} C_DIS
LIN {X 0.019,Y -551.169,Z 634.591,A 0.000,B 0.000,C 90.000,E1 322.396} C_DIS
LIN {X -0.129,Y -562.531,Z 634.586,A 0.000,B 0.000,C 90.000,E1 321.457} C_DIS
LIN {X -0.254,Y -569.424,Z 634.583,A 0.000,B 0.000,C 90.000,E1 320.884} C_DIS
LIN {X 0.010,Y -580.422,Z 634.577,A 0.000,B 0.000,C 90.000,E1 319.908} C_DIS
LIN {X 0.093,Y -588.542,Z 634.573,A 0.000,B 0.000,C 90.000,E1 319.175} C_DIS
LIN {X 0.013,Y -596.522,Z 634.569,A 0.000,B 0.000,C 90.000,E1 318.447} C_DIS
LIN {X 0.120,Y -600.330,Z 634.567,A 0.000,B 0.000,C 90.000,E1 318.081} C_DIS
LIN {X 0.335,Y -607.821,Z 634.563,A 0.000,B 0.000,C 90.000,E1 317.310} C_DIS
LIN {X 0.053,Y -612.599,Z 634.560,A 0.000,B 0.000,C 90.000,E1 316.824} C_DIS
LIN {X -0.357,Y -618.255,Z 634.557,A 0.000,B 0.000,C 90.000,E1 316.215} C_DIS
LIN {X 0.210,Y -622.503,Z 634.554,A 0.000,B 0.000,C 90.000,E1 315.648} C_DIS
LIN {X 0.180,Y -629.461,Z 634.549,A 0.000,B 0.000,C 90.000,E1 314.757} C_DIS
LIN {X 0.337,Y -634.126,Z 634.545,A 0.000,B 0.000,C 90.000,E1 314.109} C_DIS
LIN {X -0.001,Y -640.518,Z 634.540,A 0.000,B 0.000,C 90.000,E1 313.257} C_DIS
LIN {X -0.235,Y -648.361,Z 634.534,A 0.000,B 0.000,C 90.000,E1 312.162} C_DIS
LIN {X 0.073,Y -653.343,Z 634.530,A 0.000,B 0.000,C 90.000,E1 311.391} C_DIS
LIN {X -0.002,Y -656.488,Z 634.527,A 0.000,B 0.000,C 90.000,E1 310.906} C_DIS
LIN {X -0.044,Y -660.150,Z 634.524,A 0.000,B 0.000,C 90.000,E1 310.297} C_DIS
LIN {X -0.081,Y -663.463,Z 634.521,A 0.000,B 0.000,C 90.000,E1 309.688} C_DIS
LIN {X 0.001,Y -666.562,Z 634.517,A 0.000,B 0.000,C 90.000,E1 309.072} C_DIS
LIN {X -0.034,Y -668.815,Z 634.514,A 0.000,B 0.000,C 90.000,E1 308.588} C_DIS
LIN {X 0.150,Y -673.005,Z 634.509,A 0.000,B 0.000,C 90.000,E1 307.604} C_DIS
LIN {X -0.139,Y -676.616,Z 634.504,A 0.000,B 0.000,C 90.000,E1 306.664} C_DIS
LIN {X 0.006,Y -678.342,Z 634.501,A 0.000,B 0.000,C 90.000,E1 306.171} C_DIS
LIN {X -0.054,Y -682.358,Z 634.494,A 0.000,B 0.000,C 90.000,E1 304.978} C_DIS
LIN {X -0.055,Y -686.035,Z 634.488,A 0.000,B 0.000,C 90.000,E1 303.785} C_DIS
LIN {X -0.011,Y -689.490,Z 634.481,A 0.000,B 0.000,C 90.000,E1 302.594} C_DIS
LIN {X -0.069,Y -692.746,Z 634.475,A 0.000,B 0.000,C 90.000,E1 301.416} C_DIS
LIN {X 0.298,Y -695.886,Z 634.468,A 0.000,B 0.000,C 90.000,E1 300.207} C_DIS
LIN {X 0.016,Y -699.185,Z 634.460,A 0.000,B 0.000,C 90.000,E1 298.821} C_DIS
LIN {X 0.129,Y -701.630,Z 634.454,A 0.000,B 0.000,C 90.000,E1 297.641} C_DIS
LIN {X 0.015,Y -702.948,Z 634.450,A 0.000,B 0.000,C 90.000,E1 296.950} C_DIS
LIN {X 0.234,Y -703.934,Z 634.446,A 0.000,B 0.000,C 90.000,E1 296.232} C_DIS
LIN {X -0.137,Y -704.135,Z 634.443,A 0.000,B 0.000,C 90.000,E1 295.796} C_DIS
LIN {X 0.149,Y -704.118,Z 634.442,A 0.000,B 0.000,C 90.000,E1 295.540} C_DIS
LIN {X 0.084,Y -703.067,Z 634.439,A 0.000,B 0.000,C 90.000,E1 295.079} C_DIS
LIN {X 0.069,Y -702.340,Z 634.438,A 0.000,B 0.000,C 90.000,E1 294.847} C_DIS
LIN {X -0.287,Y -700.744,Z 634.437,A 0.000,B 0.000,C 90.000,E1 294.643} C_DIS
LIN {X 0.121,Y -698.055,Z 634.435,A 0.000,B 0.000,C 90.000,E1 294.259} C_DIS
LIN {X -0.031,Y -696.808,Z 634.434,A 0.000,B 0.000,C 90.000,E1 294.155} C_DIS
LIN {X 0.139,Y -694.902,Z 634.434,A 0.000,B 0.000,C 90.000,E1 294.027} C_DIS
LIN {X 0.426,Y -690.106,Z 634.433,A 0.000,B 0.000,C 90.000,E1 293.823} C_DIS
LIN {X -0.406,Y -686.381,Z 634.432,A 0.000,B 0.000,C 90.000,E1 293.770} C_DIS
LIN {X -0.125,Y -682.508,Z 634.431,A 0.000,B 0.000,C 90.000,E1 293.643} C_DIS
LIN {X 0.120,Y -675.101,Z 634.431,A 0.000,B 0.000,C 90.000,E1 293.515} C_DIS
LIN {X 0.195,Y -663.866,Z 634.430,A 0.000,B 0.000,C 90.000,E1 293.387} C_DIS
LIN {X -0.022,Y -649.886,Z 634.429,A 0.000,B 0.000,C 90.000,E1 293.206} C_DIS
LIN {X 0.035,Y -639.744,Z 634.428,A 0.000,B 0.000,C 90.000,E1 293.025} C_DIS
LIN {X -0.044,Y -630.155,Z 634.427,A 0.000,B 0.000,C 90.000,E1 292.823} C_DIS
LIN {X 0.133,Y -616.828,Z 634.425,A 0.000,B 0.000,C 90.000,E1 292.461} C_DIS
LIN {X -0.015,Y -599.879,Z 634.422,A 0.000,B 0.000,C 90.000,E1 291.972} C_DIS
LIN {X 0.144,Y -582.455,Z 634.419,A 0.000,B 0.000,C 90.000,E1 291.408} C_DIS
LIN {X -0.248,Y -577.003,Z 634.418,A 0.000,B 0.000,C 90.000,E1 291.280} C_DIS
LIN {X -0.113,Y -565.000,Z 634.416,A 0.000,B 0.000,C 90.000,E1 290.918} C_DIS
LIN {X -0.111,Y -560.720,Z 634.415,A 0.000,B 0.000,C 90.000,E1 290.737} C_DIS
LIN {X -0.115,Y -559.286,Z 634.415,A 0.000,B 0.000,C 90.000,E1 290.663} C_DIS
LIN {X -0.191,Y -556.835,Z 634.414,A 0.000,B 0.000,C 90.000,E1 290.482} C_DIS
LIN {X -0.224,Y -556.809,Z 634.414,A 0.000,B 0.000,C 90.000,E1 290.482} C_DIS
LIN {X -0.043,Y -556.126,Z 634.413,A 0.000,B 0.000,C 90.000,E1 290.301} C_DIS
LIN {X -0.020,Y -555.694,Z 634.410,A 0.000,B 0.000,C 90.000,E1 289.812} C_DIS
LIN {X 0.136,Y -555.886,Z 634.405,A 0.000,B 0.000,C 90.000,E1 288.960} C_DIS
LIN {X -0.126,Y -555.820,Z 634.399,A 0.000,B 0.000,C 90.000,E1 287.873} C_DIS
LIN {X 0.139,Y -555.559,Z 634.393,A 0.000,B 0.000,C 90.000,E1 286.732} C_DIS
LIN {X 0.244,Y -555.242,Z 634.387,A 0.000,B 0.000,C 90.000,E1 285.607} C_DIS
LIN {X -0.061,Y -554.629,Z 634.379,A 0.000,B 0.000,C 90.000,E1 284.245} C_DIS
LIN {X -0.131,Y -553.598,Z 634.368,A 0.000,B 0.000,C 90.000,E1 282.299} C_DIS
LIN {X 0.188,Y -552.642,Z 634.357,A 0.000,B 0.000,C 90.000,E1 280.310} C_DIS
LIN {X -0.254,Y -551.861,Z 634.347,A 0.000,B 0.000,C 90.000,E1 278.398} C_DIS
LIN {X 0.230,Y -551.256,Z 634.339,A 0.000,B 0.000,C 90.000,E1 276.947} C_DIS
LIN {X 0.170,Y -550.645,Z 634.328,A 0.000,B 0.000,C 90.000,E1 274.992} C_DIS
LIN {X 0.092,Y -550.097,Z 634.317,A 0.000,B 0.000,C 90.000,E1 273.037} C_DIS
LIN {X 0.252,Y -549.900,Z 634.312,A 0.000,B 0.000,C 90.000,E1 272.178} C_DIS
LIN {X 0.045,Y -549.417,Z 634.303,A 0.000,B 0.000,C 90.000,E1 270.516} C_DIS
LIN {X 0.207,Y -549.086,Z 634.298,A 0.000,B 0.000,C 90.000,E1 269.656} C_DIS
LIN {X -0.018,Y -548.302,Z 634.289,A 0.000,B 0.000,C 90.000,E1 267.993} C_DIS
LIN {X 0.243,Y -547.660,Z 634.281,A 0.000,B 0.000,C 90.000,E1 266.560} C_DIS
LIN {X -0.021,Y -546.882,Z 634.273,A 0.000,B 0.000,C 90.000,E1 265.179} C_DIS
LIN {X -0.274,Y -545.696,Z 634.264,A 0.000,B 0.000,C 90.000,E1 263.514} C_DIS
LIN {X -0.084,Y -545.022,Z 634.259,A 0.000,B 0.000,C 90.000,E1 262.648} C_DIS
LIN {X -0.266,Y -543.203,Z 634.250,A 0.000,B 0.000,C 90.000,E1 260.971} C_DIS
LIN {X -0.098,Y -540.442,Z 634.234,A 0.000,B 0.000,C 90.000,E1 258.117} C_DIS
LIN {X -0.008,Y -538.780,Z 634.223,A 0.000,B 0.000,C 90.000,E1 256.117} C_DIS
LIN {X -0.083,Y -537.570,Z 634.215,A 0.000,B 0.000,C 90.000,E1 254.700} C_DIS
LIN {X 0.205,Y -535.473,Z 634.204,A 0.000,B 0.000,C 90.000,E1 252.670} C_DIS
LIN {X -0.137,Y -534.086,Z 634.196,A 0.000,B 0.000,C 90.000,E1 251.275} C_DIS
LIN {X -0.213,Y -533.169,Z 634.191,A 0.000,B 0.000,C 90.000,E1 250.423} C_DIS
LIN {X -0.102,Y -531.609,Z 634.185,A 0.000,B 0.000,C 90.000,E1 249.263} C_DIS
LIN {X -0.018,Y -529.991,Z 634.178,A 0.000,B 0.000,C 90.000,E1 248.103} C_DIS
LIN {X -0.068,Y -527.674,Z 634.170,A 0.000,B 0.000,C 90.000,E1 246.666} C_DIS
LIN {X 0.151,Y -525.599,Z 634.164,A 0.000,B 0.000,C 90.000,E1 245.485} C_DIS
LIN {X 0.079,Y -523.276,Z 634.157,A 0.000,B 0.000,C 90.000,E1 244.332} C_DIS
LIN {X -0.202,Y -519.509,Z 634.148,A 0.000,B 0.000,C 90.000,E1 242.615} C_DIS
LIN {X -0.116,Y -517.046,Z 634.141,A 0.000,B 0.000,C 90.000,E1 241.435} C_DIS
LIN {X -0.064,Y -514.429,Z 634.135,A 0.000,B 0.000,C 90.000,E1 240.255} C_DIS
LIN {X 0.298,Y -512.369,Z 634.130,A 0.000,B 0.000,C 90.000,E1 239.331} C_DIS
LIN {X 0.070,Y -508.152,Z 634.120,A 0.000,B 0.000,C 90.000,E1 237.582} C_DIS
LIN {X 0.129,Y -504.443,Z 634.112,A 0.000,B 0.000,C 90.000,E1 236.087} C_DIS
LIN {X 0.214,Y -502.223,Z 634.107,A 0.000,B 0.000,C 90.000,E1 235.182} C_DIS
LIN {X -0.100,Y -497.499,Z 634.097,A 0.000,B 0.000,C 90.000,E1 233.417} C_DIS
LIN {X 0.175,Y -491.356,Z 634.083,A 0.000,B 0.000,C 90.000,E1 230.964} C_DIS
LIN {X 0.130,Y -485.370,Z 634.070,A 0.000,B 0.000,C 90.000,E1 228.528} C_DIS
LIN {X -0.023,Y -480.888,Z 634.060,A 0.000,B 0.000,C 90.000,E1 226.701} C_DIS
LIN {X -0.202,Y -477.827,Z 634.053,A 0.000,B 0.000,C 90.000,E1 225.486} C_DIS
LIN {X -0.213,Y -473.372,Z 634.042,A 0.000,B 0.000,C 90.000,E1 223.623} C_DIS
LIN {X -0.162,Y -470.567,Z 634.035,A 0.000,B 0.000,C 90.000,E1 222.366} C_DIS
LIN {X -0.043,Y -467.141,Z 634.027,A 0.000,B 0.000,C 90.000,E1 220.782} C_DIS
LIN {X 0.012,Y -463.720,Z 634.018,A 0.000,B 0.000,C 90.000,E1 219.197} C_DIS
LIN {X 0.200,Y -459.103,Z 634.005,A 0.000,B 0.000,C 90.000,E1 216.950} C_DIS
LIN {X -0.016,Y -454.752,Z 633.993,A 0.000,B 0.000,C 90.000,E1 214.739} C_DIS
LIN {X -0.290,Y -451.781,Z 633.984,A 0.000,B 0.000,C 90.000,E1 213.166} C_DIS
LIN {X -0.152,Y -448.314,Z 633.973,A 0.000,B 0.000,C 90.000,E1 211.209} C_DIS
LIN {X 0.279,Y -444.905,Z 633.963,A 0.000,B 0.000,C 90.000,E1 209.205} C_DIS
LIN {X 0.188,Y -441.381,Z 633.952,A 0.000,B 0.000,C 90.000,E1 207.257} C_DIS
LIN {X -0.051,Y -439.069,Z 633.944,A 0.000,B 0.000,C 90.000,E1 205.976} C_DIS
LIN {X -0.099,Y -436.087,Z 633.935,A 0.000,B 0.000,C 90.000,E1 204.335} C_DIS
LIN {X 0.014,Y -432.537,Z 633.924,A 0.000,B 0.000,C 90.000,E1 202.333} C_DIS
LIN {X -0.115,Y -427.954,Z 633.909,A 0.000,B 0.000,C 90.000,E1 199.685} C_DIS
LIN {X 0.183,Y -423.060,Z 633.893,A 0.000,B 0.000,C 90.000,E1 196.622} C_DIS
LIN {X 0.033,Y -420.428,Z 633.883,A 0.000,B 0.000,C 90.000,E1 194.954} C_DIS
LIN {X 0.075,Y -418.364,Z 633.876,A 0.000,B 0.000,C 90.000,E1 193.592} C_DIS
LIN {X -0.183,Y -414.713,Z 633.862,A 0.000,B 0.000,C 90.000,E1 191.243} C_DIS
LIN {X 0.115,Y -411.309,Z 633.849,A 0.000,B 0.000,C 90.000,E1 188.803} C_DIS
LIN {X -0.173,Y -408.327,Z 633.838,A 0.000,B 0.000,C 90.000,E1 186.777} C_DIS
LIN {X 0.190,Y -404.685,Z 633.822,A 0.000,B 0.000,C 90.000,E1 183.955} C_DIS
LIN {X 0.011,Y -402.301,Z 633.811,A 0.000,B 0.000,C 90.000,E1 181.892} C_DIS
LIN {X -0.003,Y -399.041,Z 633.791,A 0.000,B 0.000,C 90.000,E1 178.396} C_DIS
LIN {X 0.175,Y -396.522,Z 633.766,A 0.000,B 0.000,C 90.000,E1 173.799} C_DIS
LIN {X -0.104,Y -395.937,Z 633.754,A 0.000,B 0.000,C 90.000,E1 171.724} C_DIS
LIN {X 0.110,Y -395.496,Z 633.738,A 0.000,B 0.000,C 90.000,E1 168.870} C_DIS
LIN {X 0.001,Y -395.523,Z 633.723,A 0.000,B 0.000,C 90.000,E1 166.061} C_DIS
LIN {X 0.217,Y -395.791,Z 633.709,A 0.000,B 0.000,C 90.000,E1 163.559} C_DIS
LIN {X 0.050,Y -396.138,Z 633.699,A 0.000,B 0.000,C 90.000,E1 161.819} C_DIS
LIN {X 0.080,Y -396.588,Z 633.687,A 0.000,B 0.000,C 90.000,E1 159.699} C_DIS
LIN {X -0.121,Y -397.138,Z 633.676,A 0.000,B 0.000,C 90.000,E1 157.614} C_DIS
LIN {X -0.005,Y -397.694,Z 633.664,A 0.000,B 0.000,C 90.000,E1 155.485} C_DIS
LIN {X -0.067,Y -398.336,Z 633.652,A 0.000,B 0.000,C 90.000,E1 153.384} C_DIS
LIN {X 0.065,Y -398.927,Z 633.640,A 0.000,B 0.000,C 90.000,E1 151.257} C_DIS
LIN {X -0.181,Y -399.433,Z 633.631,A 0.000,B 0.000,C 90.000,E1 149.537} C_DIS
LIN {X -0.211,Y -399.941,Z 633.621,A 0.000,B 0.000,C 90.000,E1 147.788} C_DIS
LIN {X -0.130,Y -400.644,Z 633.609,A 0.000,B 0.000,C 90.000,E1 145.674} C_DIS
LIN {X -0.027,Y -401.641,Z 633.596,A 0.000,B 0.000,C 90.000,E1 143.210} C_DIS
LIN {X 0.021,Y -402.339,Z 633.586,A 0.000,B 0.000,C 90.000,E1 141.457} C_DIS
LIN {X 0.081,Y -402.991,Z 633.576,A 0.000,B 0.000,C 90.000,E1 139.703} C_DIS
LIN {X -0.200,Y -403.584,Z 633.567,A 0.000,B 0.000,C 90.000,E1 138.000} C_DIS
LIN {X -0.066,Y -404.311,Z 633.555,A 0.000,B 0.000,C 90.000,E1 135.891} C_DIS
LIN {X 0.241,Y -404.915,Z 633.545,A 0.000,B 0.000,C 90.000,E1 134.109} C_DIS
LIN {X -0.220,Y -406.598,Z 633.526,A 0.000,B 0.000,C 90.000,E1 130.701} C_DIS
LIN {X 0.044,Y -407.771,Z 633.518,A 0.000,B 0.000,C 90.000,E1 129.277} C_DIS
LIN {X 0.192,Y -408.156,Z 633.516,A 0.000,B 0.000,C 90.000,E1 128.910} C_DIS
LIN {X -0.165,Y -409.722,Z 633.512,A 0.000,B 0.000,C 90.000,E1 128.096} C_DIS
LIN {X -0.153,Y -411.957,Z 633.508,A 0.000,B 0.000,C 90.000,E1 127.443} C_DIS
LIN {X -0.216,Y -413.523,Z 633.507,A 0.000,B 0.000,C 90.000,E1 127.237} C_DIS
LIN {X -0.006,Y -415.035,Z 633.505,A 0.000,B 0.000,C 90.000,E1 126.950} C_DIS
LIN {X -0.221,Y -419.409,Z 633.503,A 0.000,B 0.000,C 90.000,E1 126.583} C_DIS
LIN {X 0.189,Y -425.892,Z 633.501,A 0.000,B 0.000,C 90.000,E1 126.091} C_DIS
LIN {X -0.063,Y -447.622,Z 633.493,A 0.000,B 0.000,C 90.000,E1 124.818} C_DIS
LIN {X 0.073,Y -457.531,Z 633.490,A 0.000,B 0.000,C 90.000,E1 124.199} C_DIS
LIN {X -0.062,Y -470.397,Z 633.485,A 0.000,B 0.000,C 90.000,E1 123.372} C_DIS
LIN {X 0.018,Y -479.901,Z 633.482,A 0.000,B 0.000,C 90.000,E1 122.704} C_DIS
LIN {X 0.010,Y -486.075,Z 633.479,A 0.000,B 0.000,C 90.000,E1 122.260} C_DIS
LIN {X -0.114,Y -495.182,Z 633.475,A 0.000,B 0.000,C 90.000,E1 121.592} C_DIS
LIN {X 0.013,Y -505.511,Z 633.471,A 0.000,B 0.000,C 90.000,E1 120.747} C_DIS
LIN {X 0.230,Y -512.457,Z 633.468,A 0.000,B 0.000,C 90.000,E1 120.129} C_DIS
LIN {X -0.139,Y -521.097,Z 633.463,A 0.000,B 0.000,C 90.000,E1 119.411} C_DIS
LIN {X 0.084,Y -530.697,Z 633.458,A 0.000,B 0.000,C 90.000,E1 118.487} C_DIS
LIN {X -0.100,Y -535.878,Z 633.455,A 0.000,B 0.000,C 90.000,E1 117.975} C_DIS
LIN {X 0.228,Y -540.901,Z 633.452,A 0.000,B 0.000,C 90.000,E1 117.385} C_DIS
LIN {X 0.159,Y -545.301,Z 633.449,A 0.000,B 0.000,C 90.000,E1 116.873} C_DIS
LIN {X -0.218,Y -548.487,Z 633.447,A 0.000,B 0.000,C 90.000,E1 116.488} C_DIS
LIN {X 0.152,Y -549.591,Z 633.446,A 0.000,B 0.000,C 90.000,E1 116.309} C_DIS
LIN {X 0.305,Y -554.156,Z 633.442,A 0.000,B 0.000,C 90.000,E1 115.591} C_DIS
LIN {X 0.257,Y -558.210,Z 633.439,A 0.000,B 0.000,C 90.000,E1 114.899} C_DIS
LIN {X 0.144,Y -562.448,Z 633.434,A 0.000,B 0.000,C 90.000,E1 114.079} C_DIS
LIN {X 0.167,Y -565.739,Z 633.430,A 0.000,B 0.000,C 90.000,E1 113.387} C_DIS
LIN {X -0.283,Y -570.380,Z 633.424,A 0.000,B 0.000,C 90.000,E1 112.333} C_DIS
LIN {X 0.242,Y -573.557,Z 633.419,A 0.000,B 0.000,C 90.000,E1 111.461} C_DIS
LIN {X 0.056,Y -576.437,Z 633.415,A 0.000,B 0.000,C 90.000,E1 110.663} C_DIS
LIN {X 0.062,Y -578.292,Z 633.412,A 0.000,B 0.000,C 90.000,E1 110.120} C_DIS
LIN {X -0.077,Y -580.808,Z 633.407,A 0.000,B 0.000,C 90.000,E1 109.322} C_DIS
LIN {X 0.012,Y -583.737,Z 633.401,A 0.000,B 0.000,C 90.000,E1 108.236} C_DIS
LIN {X -0.031,Y -586.340,Z 633.395,A 0.000,B 0.000,C 90.000,E1 107.166} C_DIS
LIN {X 0.170,Y -591.404,Z 633.384,A 0.000,B 0.000,C 90.000,E1 105.009} C_DIS
LIN {X 0.210,Y -595.352,Z 633.375,A 0.000,B 0.000,C 90.000,E1 103.411} C_DIS
LIN {X -0.102,Y -598.670,Z 633.367,A 0.000,B 0.000,C 90.000,E1 102.119} C_DIS
LIN {X 0.109,Y -601.989,Z 633.360,A 0.000,B 0.000,C 90.000,E1 100.782} C_DIS
LIN {X 0.114,Y -605.747,Z 633.351,A 0.000,B 0.000,C 90.000,E1 99.208} C_DIS
LIN {X -0.237,Y -608.701,Z 633.344,A 0.000,B 0.000,C 90.000,E1 97.936} C_DIS
LIN {X -0.196,Y -610.890,Z 633.338,A 0.000,B 0.000,C 90.000,E1 96.891} C_DIS
LIN {X 0.073,Y -613.415,Z 633.331,A 0.000,B 0.000,C 90.000,E1 95.568} C_DIS
LIN {X -0.241,Y -614.719,Z 633.327,A 0.000,B 0.000,C 90.000,E1 94.821} C_DIS
LIN {X -0.214,Y -617.208,Z 633.318,A 0.000,B 0.000,C 90.000,E1 93.269} C_DIS
LIN {X -0.184,Y -618.579,Z 633.312,A 0.000,B 0.000,C 90.000,E1 92.236} C_DIS
LIN {X -0.142,Y -619.795,Z 633.307,A 0.000,B 0.000,C 90.000,E1 91.203} C_DIS
LIN {X -0.099,Y -620.684,Z 633.301,A 0.000,B 0.000,C 90.000,E1 90.172} C_DIS
LIN {X 0.252,Y -621.200,Z 633.297,A 0.000,B 0.000,C 90.000,E1 89.370} C_DIS
LIN {X -0.311,Y -621.683,Z 633.291,A 0.000,B 0.000,C 90.000,E1 88.396} C_DIS
LIN {X -0.229,Y -621.848,Z 633.285,A 0.000,B 0.000,C 90.000,E1 87.364} C_DIS
LIN {X 0.180,Y -621.688,Z 633.278,A 0.000,B 0.000,C 90.000,E1 86.045} C_DIS
LIN {X 0.310,Y -621.281,Z 633.272,A 0.000,B 0.000,C 90.000,E1 85.008} C_DIS
LIN {X 0.133,Y -620.581,Z 633.265,A 0.000,B 0.000,C 90.000,E1 83.742} C_DIS
LIN {X 0.015,Y -619.570,Z 633.258,A 0.000,B 0.000,C 90.000,E1 82.470} C_DIS
LIN {X -0.256,Y -618.744,Z 633.254,A 0.000,B 0.000,C 90.000,E1 81.724} C_DIS
LIN {X -0.079,Y -617.397,Z 633.248,A 0.000,B 0.000,C 90.000,E1 80.679} C_DIS
LIN {X 0.079,Y -615.934,Z 633.242,A 0.000,B 0.000,C 90.000,E1 79.634} C_DIS
LIN {X 0.091,Y -613.780,Z 633.235,A 0.000,B 0.000,C 90.000,E1 78.342} C_DIS
LIN {X 0.188,Y -611.916,Z 633.230,A 0.000,B 0.000,C 90.000,E1 77.297} C_DIS
LIN {X 0.276,Y -609.340,Z 633.222,A 0.000,B 0.000,C 90.000,E1 75.992} C_DIS
LIN {X 0.171,Y -606.618,Z 633.215,A 0.000,B 0.000,C 90.000,E1 74.700} C_DIS
LIN {X 0.340,Y -603.586,Z 633.208,A 0.000,B 0.000,C 90.000,E1 73.378} C_DIS
LIN {X -0.291,Y -600.391,Z 633.201,A 0.000,B 0.000,C 90.000,E1 72.127} C_DIS
LIN {X -0.206,Y -598.226,Z 633.196,A 0.000,B 0.000,C 90.000,E1 71.329} C_DIS
LIN {X 0.228,Y -595.782,Z 633.192,A 0.000,B 0.000,C 90.000,E1 70.496} C_DIS
LIN {X -0.181,Y -594.116,Z 633.189,A 0.000,B 0.000,C 90.000,E1 70.007} C_DIS
LIN {X 0.285,Y -590.349,Z 633.183,A 0.000,B 0.000,C 90.000,E1 68.901} C_DIS
LIN {X -0.157,Y -588.354,Z 633.180,A 0.000,B 0.000,C 90.000,E1 68.411} C_DIS
LIN {X -0.315,Y -583.957,Z 633.174,A 0.000,B 0.000,C 90.000,E1 67.358} C_DIS
LIN {X 0.230,Y -579.223,Z 633.168,A 0.000,B 0.000,C 90.000,E1 66.230} C_DIS
LIN {X -0.068,Y -574.026,Z 633.162,A 0.000,B 0.000,C 90.000,E1 65.177} C_DIS
LIN {X -0.305,Y -571.963,Z 633.160,A 0.000,B 0.000,C 90.000,E1 64.793} C_DIS
LIN {X 0.045,Y -568.172,Z 633.156,A 0.000,B 0.000,C 90.000,E1 64.076} C_DIS
LIN {X 0.201,Y -564.952,Z 633.153,A 0.000,B 0.000,C 90.000,E1 63.512} C_DIS
LIN {X 0.043,Y -559.688,Z 633.149,A 0.000,B 0.000,C 90.000,E1 62.743} C_DIS
LIN {X -0.361,Y -555.638,Z 633.146,A 0.000,B 0.000,C 90.000,E1 62.231} C_DIS
LIN {X 0.296,Y -551.603,Z 633.143,A 0.000,B 0.000,C 90.000,E1 61.641} C_DIS
LIN {X -0.111,Y -546.581,Z 633.140,A 0.000,B 0.000,C 90.000,E1 61.129} C_DIS
LIN {X -0.088,Y -543.755,Z 633.138,A 0.000,B 0.000,C 90.000,E1 60.845} C_DIS
LIN {X -0.066,Y -541.921,Z 633.137,A 0.000,B 0.000,C 90.000,E1 60.639} C_DIS
LIN {X 0.090,Y -536.261,Z 633.134,A 0.000,B 0.000,C 90.000,E1 60.127} C_DIS
LIN {X 0.097,Y -530.196,Z 633.132,A 0.000,B 0.000,C 90.000,E1 59.665} C_DIS
LIN {X 0.063,Y -525.310,Z 633.130,A 0.000,B 0.000,C 90.000,E1 59.331} C_DIS
LIN {X -0.025,Y -518.962,Z 633.128,A 0.000,B 0.000,C 90.000,E1 58.948} C_DIS
LIN {X -0.043,Y -513.897,Z 633.126,A 0.000,B 0.000,C 90.000,E1 58.663} C_DIS
LIN {X -0.237,Y -507.128,Z 633.124,A 0.000,B 0.000,C 90.000,E1 58.329} C_DIS
LIN {X -0.047,Y -490.280,Z 633.119,A 0.000,B 0.000,C 90.000,E1 57.454} C_DIS
LIN {X 0.079,Y -470.216,Z 633.114,A 0.000,B 0.000,C 90.000,E1 56.421} C_DIS
LIN {X 0.029,Y -445.069,Z 633.106,A 0.000,B 0.000,C 90.000,E1 55.102} C_DIS
LIN {X 0.078,Y -439.857,Z 633.105,A 0.000,B 0.000,C 90.000,E1 54.815} C_DIS
LIN {X 0.034,Y -439.767,Z 633.105,A 0.000,B 0.000,C 90.000,E1 54.815} C_DIS
LIN {X 0.042,Y -431.868,Z 633.083,A 0.000,B 0.000,C 90.000,E1 51.009} C_DIS
LIN {X 0.028,Y -431.185,Z 633.082,A 0.000,B 0.000,C 90.000,E1 50.678} C_DIS
LIN {X -0.231,Y -424.959,Z 633.067,A 0.000,B 0.000,C 90.000,E1 48.081} C_DIS
LIN {X 0.000,Y -425.554,Z 633.059,A 0.000,B 0.000,C 90.000,E1 46.662} C_DIS
LIN {X -0.227,Y -426.003,Z 633.048,A 0.000,B 0.000,C 90.000,E1 44.676} C_DIS
LIN {X -0.023,Y -426.736,Z 633.033,A 0.000,B 0.000,C 90.000,E1 41.962} C_DIS
LIN {X 0.117,Y -427.510,Z 633.022,A 0.000,B 0.000,C 90.000,E1 39.930} C_DIS
LIN {X 0.004,Y -428.407,Z 633.011,A 0.000,B 0.000,C 90.000,E1 37.935} C_DIS
LIN {X -0.015,Y -429.401,Z 633.000,A 0.000,B 0.000,C 90.000,E1 35.931} C_DIS
LIN {X 0.089,Y -430.288,Z 632.989,A 0.000,B 0.000,C 90.000,E1 33.913} C_DIS
LIN {X -0.029,Y -430.884,Z 632.979,A 0.000,B 0.000,C 90.000,E1 32.260} C_DIS
LIN {X -0.003,Y -431.523,Z 632.970,A 0.000,B 0.000,C 90.000,E1 30.590} C_DIS
LIN {X -0.169,Y -432.337,Z 632.959,A 0.000,B 0.000,C 90.000,E1 28.615} C_DIS
LIN {X 0.048,Y -433.032,Z 632.950,A 0.000,B 0.000,C 90.000,E1 26.924} C_DIS
LIN {X -0.108,Y -433.840,Z 632.940,A 0.000,B 0.000,C 90.000,E1 25.283} C_DIS
LIN {X -0.021,Y -434.972,Z 632.928,A 0.000,B 0.000,C 90.000,E1 22.950} C_DIS
LIN {X 0.261,Y -435.762,Z 632.920,A 0.000,B 0.000,C 90.000,E1 21.589} C_DIS
LIN {X -0.179,Y -436.707,Z 632.911,A 0.000,B 0.000,C 90.000,E1 19.993} C_DIS
LIN {X -0.091,Y -437.766,Z 632.900,A 0.000,B 0.000,C 90.000,E1 18.000} C_DIS
LIN {X 0.145,Y -439.133,Z 632.887,A 0.000,B 0.000,C 90.000,E1 15.662} C_DIS
LIN {X -0.099,Y -440.853,Z 632.873,A 0.000,B 0.000,C 90.000,E1 13.063} C_DIS
LIN {X 0.067,Y -442.420,Z 632.862,A 0.000,B 0.000,C 90.000,E1 11.074} C_DIS
LIN {X -0.178,Y -444.985,Z 632.845,A 0.000,B 0.000,C 90.000,E1 8.163} C_DIS
LIN {X -0.129,Y -446.943,Z 632.834,A 0.000,B 0.000,C 90.000,E1 6.201} C_DIS
LIN {X -0.197,Y -449.770,Z 632.820,A 0.000,B 0.000,C 90.000,E1 3.612} C_DIS
LIN {X 0.159,Y -451.736,Z 632.811,A 0.000,B 0.000,C 90.000,E1 1.949} C_DIS
LIN {X -0.204,Y -455.991,Z 632.794,A 0.000,B 0.000,C 90.000,E1 358.854} C_DIS
LIN {X 0.223,Y -459.480,Z 632.781,A 0.000,B 0.000,C 90.000,E1 356.560} C_DIS
LIN {X -0.137,Y -463.204,Z 632.769,A 0.000,B 0.000,C 90.000,E1 354.375} C_DIS
LIN {X -0.103,Y -466.444,Z 632.758,A 0.000,B 0.000,C 90.000,E1 352.470} C_DIS
LIN {X 0.074,Y -469.773,Z 632.748,A 0.000,B 0.000,C 90.000,E1 350.557} C_DIS
LIN {X 0.024,Y -472.415,Z 632.739,A 0.000,B 0.000,C 90.000,E1 348.993} C_DIS
LIN {X 0.036,Y -475.664,Z 632.729,A 0.000,B 0.000,C 90.000,E1 347.117} C_DIS
LIN {X 0.052,Y -480.124,Z 632.715,A 0.000,B 0.000,C 90.000,E1 344.629} C_DIS
LIN {X 0.021,Y -483.612,Z 632.704,A 0.000,B 0.000,C 90.000,E1 342.779} C_DIS
LIN {X -0.270,Y -486.041,Z 632.698,A 0.000,B 0.000,C 90.000,E1 341.583} C_DIS
LIN {X 0.127,Y -489.625,Z 632.687,A 0.000,B 0.000,C 90.000,E1 339.699} C_DIS
LIN {X -0.130,Y -493.139,Z 632.677,A 0.000,B 0.000,C 90.000,E1 337.901} C_DIS
LIN {X 0.002,Y -494.737,Z 632.672,A 0.000,B 0.000,C 90.000,E1 336.975} C_DIS
LIN {X -0.203,Y -497.227,Z 632.664,A 0.000,B 0.000,C 90.000,E1 335.485} C_DIS
LIN {X 0.053,Y -499.541,Z 632.655,A 0.000,B 0.000,C 90.000,E1 333.948} C_DIS
LIN {X -0.023,Y -502.297,Z 632.645,A 0.000,B 0.000,C 90.000,E1 332.153} C_DIS
LIN {X -0.050,Y -507.659,Z 632.627,A 0.000,B 0.000,C 90.000,E1 328.869} C_DIS
LIN {X 0.125,Y -509.998,Z 632.620,A 0.000,B 0.000,C 90.000,E1 327.661} C_DIS
LIN {X -0.008,Y -512.222,Z 632.616,A 0.000,B 0.000,C 90.000,E1 326.786} C_DIS
LIN {X 0.349,Y -514.471,Z 632.611,A 0.000,B 0.000,C 90.000,E1 326.008} C_DIS
LIN {X -0.045,Y -517.190,Z 632.608,A 0.000,B 0.000,C 90.000,E1 325.435} C_DIS
LIN {X 0.185,Y -519.085,Z 632.606,A 0.000,B 0.000,C 90.000,E1 325.102} C_DIS
LIN {X 0.004,Y -519.810,Z 632.605,A 0.000,B 0.000,C 90.000,E1 324.975} C_DIS
LIN {X -0.104,Y -524.311,Z 632.602,A 0.000,B 0.000,C 90.000,E1 324.402} C_DIS
LIN {X -0.097,Y -528.381,Z 632.600,A 0.000,B 0.000,C 90.000,E1 323.989} C_DIS
LIN {X 0.005,Y -534.318,Z 632.597,A 0.000,B 0.000,C 90.000,E1 323.463} C_DIS
LIN {X 0.019,Y -543.071,Z 632.593,A 0.000,B 0.000,C 90.000,E1 322.763} C_DIS
LIN {X -0.246,Y -550.247,Z 632.590,A 0.000,B 0.000,C 90.000,E1 322.190} C_DIS
LIN {X -0.010,Y -563.158,Z 632.584,A 0.000,B 0.000,C 90.000,E1 321.090} C_DIS
LIN {X 0.214,Y -571.587,Z 632.580,A 0.000,B 0.000,C 90.000,E1 320.356} C_DIS
LIN {X 0.002,Y -581.331,Z 632.575,A 0.000,B 0.000,C 90.000,E1 319.542} C_DIS
LIN {X 0.075,Y -590.816,Z 632.571,A 0.000,B 0.000,C 90.000,E1 318.690} C_DIS
LIN {X 0.090,Y -598.791,Z 632.567,A 0.000,B 0.000,C 90.000,E1 317.957} C_DIS
LIN {X 0.386,Y -605.100,Z 632.563,A 0.000,B 0.000,C 90.000,E1 317.310} C_DIS
LIN {X -0.195,Y -608.773,Z 632.561,A 0.000,B 0.000,C 90.000,E1 316.986} C_DIS
LIN {X -0.101,Y -613.526,Z 632.558,A 0.000,B 0.000,C 90.000,E1 316.458} C_DIS
LIN {X 0.078,Y -616.961,Z 632.556,A 0.000,B 0.000,C 90.000,E1 316.053} C_DIS
LIN {X 0.275,Y -620.272,Z 632.554,A 0.000,B 0.000,C 90.000,E1 315.648} C_DIS
LIN {X -0.157,Y -626.447,Z 632.549,A 0.000,B 0.000,C 90.000,E1 314.919} C_DIS
LIN {X -0.029,Y -631.322,Z 632.546,A 0.000,B 0.000,C 90.000,E1 314.271} C_DIS
LIN {X 0.048,Y -638.709,Z 632.540,A 0.000,B 0.000,C 90.000,E1 313.257} C_DIS
LIN {X 0.200,Y -645.022,Z 632.536,A 0.000,B 0.000,C 90.000,E1 312.366} C_DIS
LIN {X 0.045,Y -649.349,Z 632.532,A 0.000,B 0.000,C 90.000,E1 311.757} C_DIS
LIN {X -0.099,Y -655.141,Z 632.527,A 0.000,B 0.000,C 90.000,E1 310.906} C_DIS
LIN {X -0.157,Y -659.642,Z 632.523,A 0.000,B 0.000,C 90.000,E1 310.172} C_DIS
LIN {X -0.194,Y -662.975,Z 632.520,A 0.000,B 0.000,C 90.000,E1 309.564} C_DIS
LIN {X 0.269,Y -665.509,Z 632.517,A 0.000,B 0.000,C 90.000,E1 309.036} C_DIS
LIN {X 0.288,Y -667.298,Z 632.515,A 0.000,B 0.000,C 90.000,E1 308.669} C_DIS
LIN {X -0.076,Y -671.546,Z 632.510,A 0.000,B 0.000,C 90.000,E1 307.729} C_DIS
LIN {X 0.030,Y -673.505,Z 632.507,A 0.000,B 0.000,C 90.000,E1 307.237} C_DIS
LIN {X -0.255,Y -677.187,Z 632.502,A 0.000,B 0.000,C 90.000,E1 306.297} C_DIS
LIN {X -0.342,Y -681.253,Z 632.495,A 0.000,B 0.000,C 90.000,E1 305.105} C_DIS
LIN {X 0.205,Y -684.995,Z 632.488,A 0.000,B 0.000,C 90.000,E1 303.865} C_DIS
LIN {X 0.238,Y -688.519,Z 632.482,A 0.000,B 0.000,C 90.000,E1 302.673} C_DIS
LIN {X -0.059,Y -691.256,Z 632.476,A 0.000,B 0.000,C 90.000,E1 301.750} C_DIS
LIN {X -0.070,Y -695.134,Z 632.469,A 0.000,B 0.000,C 90.000,E1 300.335} C_DIS
LIN {X -0.178,Y -696.331,Z 632.466,A 0.000,B 0.000,C 90.000,E1 299.873} C_DIS
LIN {X -0.106,Y -699.123,Z 632.459,A 0.000,B 0.000,C 90.000,E1 298.693} C_DIS
LIN {X 0.004,Y -701.636,Z 632.453,A 0.000,B 0.000,C 90.000,E1 297.513} C_DIS
LIN {X -0.107,Y -702.908,Z 632.449,A 0.000,B 0.000,C 90.000,E1 296.821} C_DIS
LIN {X -0.174,Y -703.595,Z 632.446,A 0.000,B 0.000,C 90.000,E1 296.360} C_DIS
LIN {X -0.261,Y -703.981,Z 632.443,A 0.000,B 0.000,C 90.000,E1 295.668} C_DIS
LIN {X 0.025,Y -703.584,Z 632.441,A 0.000,B 0.000,C 90.000,E1 295.412} C_DIS
LIN {X -0.045,Y -702.492,Z 632.439,A 0.000,B 0.000,C 90.000,E1 294.951} C_DIS
LIN {X 0.095,Y -701.970,Z 632.438,A 0.000,B 0.000,C 90.000,E1 294.823} C_DIS
LIN {X -0.285,Y -698.489,Z 632.435,A 0.000,B 0.000,C 90.000,E1 294.387} C_DIS
LIN {X -0.150,Y -697.501,Z 632.435,A 0.000,B 0.000,C 90.000,E1 294.259} C_DIS
LIN {X -0.019,Y -696.093,Z 632.434,A 0.000,B 0.000,C 90.000,E1 294.131} C_DIS
LIN {X -0.171,Y -693.743,Z 632.433,A 0.000,B 0.000,C 90.000,E1 294.027} C_DIS
LIN {X 0.385,Y -689.449,Z 632.433,A 0.000,B 0.000,C 90.000,E1 293.823} C_DIS
LIN {X -0.407,Y -685.832,Z 632.432,A 0.000,B 0.000,C 90.000,E1 293.770} C_DIS
LIN {X -0.220,Y -681.389,Z 632.431,A 0.000,B 0.000,C 90.000,E1 293.643} C_DIS
LIN {X 0.023,Y -673.443,Z 632.431,A 0.000,B 0.000,C 90.000,E1 293.515} C_DIS
LIN {X -0.088,Y -667.020,Z 632.430,A 0.000,B 0.000,C 90.000,E1 293.462} C_DIS
LIN {X 0.185,Y -653.620,Z 632.429,A 0.000,B 0.000,C 90.000,E1 293.259} C_DIS
LIN {X -0.338,Y -640.128,Z 632.428,A 0.000,B 0.000,C 90.000,E1 293.078} C_DIS
LIN {X 0.192,Y -630.474,Z 632.427,A 0.000,B 0.000,C 90.000,E1 292.823} C_DIS
LIN {X 0.058,Y -620.803,Z 632.426,A 0.000,B 0.000,C 90.000,E1 292.589} C_DIS
LIN {X 0.264,Y -603.741,Z 632.423,A 0.000,B 0.000,C 90.000,E1 292.078} C_DIS
LIN {X 0.248,Y -586.427,Z 632.420,A 0.000,B 0.000,C 90.000,E1 291.535} C_DIS
LIN {X 0.035,Y -577.533,Z 632.418,A 0.000,B 0.000,C 90.000,E1 291.280} C_DIS
LIN {X -0.131,Y -568.677,Z 632.417,A 0.000,B 0.000,C 90.000,E1 291.046} C_DIS
LIN {X 0.144,Y -563.938,Z 632.416,A 0.000,B 0.000,C 90.000,E1 290.865} C_DIS
LIN {X 0.119,Y -559.429,Z 632.415,A 0.000,B 0.000,C 90.000,E1 290.663} C_DIS
LIN {X -0.179,Y -556.799,Z 632.414,A 0.000,B 0.000,C 90.000,E1 290.482} C_DIS
LIN {X -0.215,Y -556.779,Z 632.414,A 0.000,B 0.000,C 90.000,E1 290.482} C_DIS
LIN {X 0.062,Y -556.374,Z 632.413,A 0.000,B 0.000,C 90.000,E1 290.355} C_DIS
LIN {X -0.031,Y -556.129,Z 632.413,A 0.000,B 0.000,C 90.000,E1 290.248} C_DIS
LIN {X 0.293,Y -555.800,Z 632.410,A 0.000,B 0.000,C 90.000,E1 289.812} C_DIS
LIN {X -0.163,Y -555.975,Z 632.406,A 0.000,B 0.000,C 90.000,E1 289.033} C_DIS
LIN {X 0.282,Y -555.937,Z 632.400,A 0.000,B 0.000,C 90.000,E1 287.873} C_DIS
LIN {X -0.143,Y -555.694,Z 632.393,A 0.000,B 0.000,C 90.000,E1 286.804} C_DIS
LIN {X 0.122,Y -555.382,Z 632.387,A 0.000,B 0.000,C 90.000,E1 285.662} C_DIS
LIN {X 0.227,Y -554.882,Z 632.381,A 0.000,B 0.000,C 90.000,E1 284.537} C_DIS
LIN {X 0.034,Y -554.032,Z 632.372,A 0.000,B 0.000,C 90.000,E1 282.883} C_DIS
LIN {X -0.180,Y -553.037,Z 632.361,A 0.000,B 0.000,C 90.000,E1 280.950} C_DIS
LIN {X -0.098,Y -552.315,Z 632.351,A 0.000,B 0.000,C 90.000,E1 279.265} C_DIS
LIN {X -0.113,Y -551.630,Z 632.342,A 0.000,B 0.000,C 90.000,E1 277.587} C_DIS
LIN {X -0.002,Y -550.796,Z 632.330,A 0.000,B 0.000,C 90.000,E1 275.334} C_DIS
LIN {X -0.114,Y -550.238,Z 632.319,A 0.000,B 0.000,C 90.000,E1 273.383} C_DIS
LIN {X 0.130,Y -549.948,Z 632.313,A 0.000,B 0.000,C 90.000,E1 272.236} C_DIS
LIN {X -0.076,Y -549.491,Z 632.303,A 0.000,B 0.000,C 90.000,E1 270.573} C_DIS
LIN {X 0.140,Y -549.022,Z 632.297,A 0.000,B 0.000,C 90.000,E1 269.427} C_DIS
LIN {X -0.136,Y -548.383,Z 632.289,A 0.000,B 0.000,C 90.000,E1 268.051} C_DIS
LIN {X 0.128,Y -547.781,Z 632.281,A 0.000,B 0.000,C 90.000,E1 266.617} C_DIS
LIN {X -0.178,Y -547.007,Z 632.273,A 0.000,B 0.000,C 90.000,E1 265.241} C_DIS
LIN {X 0.161,Y -545.845,Z 632.264,A 0.000,B 0.000,C 90.000,E1 263.514} C_DIS
LIN {X -0.188,Y -545.196,Z 632.259,A 0.000,B 0.000,C 90.000,E1 262.704} C_DIS
LIN {X 0.171,Y -543.687,Z 632.252,A 0.000,B 0.000,C 90.000,E1 261.254} C_DIS
LIN {X -0.027,Y -542.138,Z 632.244,A 0.000,B 0.000,C 90.000,E1 259.859} C_DIS
LIN {X -0.109,Y -540.325,Z 632.233,A 0.000,B 0.000,C 90.000,E1 257.881} C_DIS
LIN {X -0.018,Y -538.688,Z 632.222,A 0.000,B 0.000,C 90.000,E1 255.880} C_DIS
LIN {X -0.154,Y -537.729,Z 632.215,A 0.000,B 0.000,C 90.000,E1 254.755} C_DIS
LIN {X 0.099,Y -535.919,Z 632.206,A 0.000,B 0.000,C 90.000,E1 253.015} C_DIS
LIN {X -0.191,Y -534.217,Z 632.196,A 0.000,B 0.000,C 90.000,E1 251.329} C_DIS
LIN {X -0.242,Y -532.937,Z 632.190,A 0.000,B 0.000,C 90.000,E1 250.188} C_DIS
LIN {X -0.139,Y -531.355,Z 632.183,A 0.000,B 0.000,C 90.000,E1 249.028} C_DIS
LIN {X 0.135,Y -529.677,Z 632.177,A 0.000,B 0.000,C 90.000,E1 247.847} C_DIS
LIN {X 0.082,Y -527.327,Z 632.169,A 0.000,B 0.000,C 90.000,E1 246.410} C_DIS
LIN {X -0.181,Y -525.154,Z 632.163,A 0.000,B 0.000,C 90.000,E1 245.281} C_DIS
LIN {X -0.164,Y -523.425,Z 632.158,A 0.000,B 0.000,C 90.000,E1 244.409} C_DIS
LIN {X 0.115,Y -520.298,Z 632.150,A 0.000,B 0.000,C 90.000,E1 242.922} C_DIS
LIN {X 0.092,Y -517.162,Z 632.142,A 0.000,B 0.000,C 90.000,E1 241.463} C_DIS
LIN {X -0.312,Y -514.549,Z 632.135,A 0.000,B 0.000,C 90.000,E1 240.333} C_DIS
LIN {X 0.049,Y -512.493,Z 632.130,A 0.000,B 0.000,C 90.000,E1 239.410} C_DIS
LIN {X -0.180,Y -508.251,Z 632.120,A 0.000,B 0.000,C 90.000,E1 237.661} C_DIS
LIN {X -0.119,Y -504.538,Z 632.112,A 0.000,B 0.000,C 90.000,E1 236.167} C_DIS
LIN {X -0.149,Y -501.523,Z 632.105,A 0.000,B 0.000,C 90.000,E1 234.975} C_DIS
LIN {X 0.220,Y -496.743,Z 632.095,A 0.000,B 0.000,C 90.000,E1 233.130} C_DIS
LIN {X -0.071,Y -491.413,Z 632.084,A 0.000,B 0.000,C 90.000,E1 231.045} C_DIS
LIN {X -0.261,Y -486.131,Z 632.072,A 0.000,B 0.000,C 90.000,E1 228.933} C_DIS
LIN {X -0.012,Y -483.139,Z 632.065,A 0.000,B 0.000,C 90.000,E1 227.676} C_DIS
LIN {X -0.010,Y -479.411,Z 632.056,A 0.000,B 0.000,C 90.000,E1 226.134} C_DIS
LIN {X 0.117,Y -474.123,Z 632.044,A 0.000,B 0.000,C 90.000,E1 223.947} C_DIS
LIN {X -0.050,Y -470.578,Z 632.036,A 0.000,B 0.000,C 90.000,E1 222.405} C_DIS
LIN {X 0.029,Y -467.162,Z 632.027,A 0.000,B 0.000,C 90.000,E1 220.825} C_DIS
LIN {X -0.217,Y -463.748,Z 632.018,A 0.000,B 0.000,C 90.000,E1 219.277} C_DIS
LIN {X -0.024,Y -459.104,Z 632.006,A 0.000,B 0.000,C 90.000,E1 217.030} C_DIS
LIN {X -0.232,Y -454.734,Z 631.993,A 0.000,B 0.000,C 90.000,E1 214.818} C_DIS
LIN {X 0.125,Y -451.796,Z 631.984,A 0.000,B 0.000,C 90.000,E1 213.166} C_DIS
LIN {X -0.125,Y -448.292,Z 631.974,A 0.000,B 0.000,C 90.000,E1 211.258} C_DIS
LIN {X 0.081,Y -444.878,Z 631.963,A 0.000,B 0.000,C 90.000,E1 209.283} C_DIS
LIN {X 0.153,Y -441.949,Z 631.954,A 0.000,B 0.000,C 90.000,E1 207.641} C_DIS
LIN {X -0.045,Y -439.065,Z 631.945,A 0.000,B 0.000,C 90.000,E1 206.027} C_DIS
LIN {X -0.097,Y -436.079,Z 631.935,A 0.000,B 0.000,C 90.000,E1 204.387} C_DIS
LIN {X 0.009,Y -432.549,Z 631.924,A 0.000,B 0.000,C 90.000,E1 202.386} C_DIS
LIN {X -0.078,Y -428.533,Z 631.911,A 0.000,B 0.000,C 90.000,E1 200.066} C_DIS
LIN {X 0.129,Y -424.656,Z 631.898,A 0.000,B 0.000,C 90.000,E1 197.692} C_DIS
LIN {X 0.006,Y -422.060,Z 631.889,A 0.000,B 0.000,C 90.000,E1 196.024} C_DIS
LIN {X -0.105,Y -418.977,Z 631.878,A 0.000,B 0.000,C 90.000,E1 194.008} C_DIS
LIN {X 0.153,Y -415.275,Z 631.865,A 0.000,B 0.000,C 90.000,E1 191.591} C_DIS
LIN {X 0.091,Y -411.391,Z 631.849,A 0.000,B 0.000,C 90.000,E1 188.859} C_DIS
LIN {X -0.197,Y -408.429,Z 631.838,A 0.000,B 0.000,C 90.000,E1 186.834} C_DIS
LIN {X 0.168,Y -404.784,Z 631.822,A 0.000,B 0.000,C 90.000,E1 184.012} C_DIS
LIN {X -0.009,Y -402.404,Z 631.811,A 0.000,B 0.000,C 90.000,E1 181.949} C_DIS
LIN {X 0.029,Y -399.417,Z 631.793,A 0.000,B 0.000,C 90.000,E1 178.797} C_DIS
LIN {X 0.166,Y -396.606,Z 631.766,A 0.000,B 0.000,C 90.000,E1 173.856} C_DIS
LIN {X -0.109,Y -396.045,Z 631.754,A 0.000,B 0.000,C 90.000,E1 171.781} C_DIS
LIN {X 0.112,Y -395.596,Z 631.739,A 0.000,B 0.000,C 90.000,E1 168.926} C_DIS
LIN {X 0.011,Y -395.645,Z 631.723,A 0.000,B 0.000,C 90.000,E1 166.117} C_DIS
LIN {X 0.171,Y -395.879,Z 631.711,A 0.000,B 0.000,C 90.000,E1 163.976} C_DIS
LIN {X 0.074,Y -396.271,Z 631.699,A 0.000,B 0.000,C 90.000,E1 161.873} C_DIS
LIN {X 0.180,Y -396.805,Z 631.686,A 0.000,B 0.000,C 90.000,E1 159.390} C_DIS
LIN {X -0.080,Y -397.280,Z 631.676,A 0.000,B 0.000,C 90.000,E1 157.667} C_DIS
LIN {X -0.179,Y -397.784,Z 631.666,A 0.000,B 0.000,C 90.000,E1 155.921} C_DIS
LIN {X 0.122,Y -398.394,Z 631.654,A 0.000,B 0.000,C 90.000,E1 153.768} C_DIS
LIN {X 0.027,Y -398.926,Z 631.645,A 0.000,B 0.000,C 90.000,E1 152.025} C_DIS
LIN {X 0.134,Y -399.451,Z 631.635,A 0.000,B 0.000,C 90.000,E1 150.255} C_DIS
LIN {X 0.222,Y -400.167,Z 631.621,A 0.000,B 0.000,C 90.000,E1 147.788} C_DIS
LIN {X -0.023,Y -400.835,Z 631.610,A 0.000,B 0.000,C 90.000,E1 145.722} C_DIS
LIN {X 0.096,Y -401.826,Z 631.596,A 0.000,B 0.000,C 90.000,E1 143.256} C_DIS
LIN {X -0.095,Y -402.517,Z 631.586,A 0.000,B 0.000,C 90.000,E1 141.537} C_DIS
LIN {X -0.033,Y -403.157,Z 631.577,A 0.000,B 0.000,C 90.000,E1 139.784} C_DIS
LIN {X 0.084,Y -403.852,Z 631.565,A 0.000,B 0.000,C 90.000,E1 137.676} C_DIS
LIN {X 0.228,Y -404.540,Z 631.553,A 0.000,B 0.000,C 90.000,E1 135.567} C_DIS
LIN {X -0.033,Y -405.107,Z 631.544,A 0.000,B 0.000,C 90.000,E1 133.866} C_DIS
LIN {X -0.060,Y -406.579,Z 631.526,A 0.000,B 0.000,C 90.000,E1 130.744} C_DIS
LIN {X -0.206,Y -407.289,Z 631.521,A 0.000,B 0.000,C 90.000,E1 129.725} C_DIS
LIN {X 0.088,Y -407.941,Z 631.517,A 0.000,B 0.000,C 90.000,E1 128.991} C_DIS
LIN {X -0.019,Y -409.270,Z 631.512,A 0.000,B 0.000,C 90.000,E1 128.141} C_DIS
LIN {X 0.022,Y -411.486,Z 631.507,A 0.000,B 0.000,C 90.000,E1 127.317} C_DIS
LIN {X 0.102,Y -414.333,Z 631.505,A 0.000,B 0.000,C 90.000,E1 126.790} C_DIS
LIN {X -0.129,Y -416.628,Z 631.503,A 0.000,B 0.000,C 90.000,E1 126.583} C_DIS
LIN {X 0.061,Y -420.777,Z 631.501,A 0.000,B 0.000,C 90.000,E1 126.217} C_DIS
LIN {X 0.016,Y -427.207,Z 631.499,A 0.000,B 0.000,C 90.000,E1 125.804} C_DIS
LIN {X 0.000,Y -447.450,Z 631.492,A 0.000,B 0.000,C 90.000,E1 124.612} C_DIS
LIN {X -0.010,Y -455.753,Z 631.490,A 0.000,B 0.000,C 90.000,E1 124.119} C_DIS
LIN {X 0.173,Y -467.068,Z 631.486,A 0.000,B 0.000,C 90.000,E1 123.372} C_DIS
LIN {X 0.104,Y -473.411,Z 631.483,A 0.000,B 0.000,C 90.000,E1 122.959} C_DIS
LIN {X 0.194,Y -484.082,Z 631.479,A 0.000,B 0.000,C 90.000,E1 122.212} C_DIS
LIN {X 0.049,Y -493.310,Z 631.475,A 0.000,B 0.000,C 90.000,E1 121.544} C_DIS
LIN {X -0.328,Y -500.802,Z 631.472,A 0.000,B 0.000,C 90.000,E1 121.003} C_DIS
LIN {X 0.192,Y -506.727,Z 631.469,A 0.000,B 0.000,C 90.000,E1 120.463} C_DIS
LIN {X 0.073,Y -512.356,Z 631.467,A 0.000,B 0.000,C 90.000,E1 120.001} C_DIS
LIN {X -0.071,Y -520.793,Z 631.463,A 0.000,B 0.000,C 90.000,E1 119.283} C_DIS
LIN {X 0.199,Y -526.373,Z 631.460,A 0.000,B 0.000,C 90.000,E1 118.743} C_DIS
LIN {X 0.115,Y -530.561,Z 631.458,A 0.000,B 0.000,C 90.000,E1 118.359} C_DIS
LIN {X -0.218,Y -535.503,Z 631.455,A 0.000,B 0.000,C 90.000,E1 117.897} C_DIS
LIN {X -0.077,Y -540.185,Z 631.452,A 0.000,B 0.000,C 90.000,E1 117.385} C_DIS
LIN {X -0.063,Y -545.049,Z 631.449,A 0.000,B 0.000,C 90.000,E1 116.821} C_DIS
LIN {X 0.176,Y -549.458,Z 631.446,A 0.000,B 0.000,C 90.000,E1 116.232} C_DIS
